	ReadStatus
	(
		pDestAddr := ADR(OUT_State),
		sIPAddr := ParamIpAddress,
		tTimeout := ParamTimeOut,
		nTcpPort := ParamTcpPort,
		nQuantity := 1,
		nMBAddr := 2,
		cbLength := SIZEOF(OUT_State),
		ClockRead := ClockRead AND MesDataExd.MesData.MesCP_Read,
		nUnitID := ParamUnitID
	);
	
	R_TrigState(CLK := OUT_State AND TpUpdate.Q);
	F_TrigState(CLK := OUT_State AND TpUpdate.Q);
	
	IF R_TrigState.Q THEN
		TimeStart := TIME();
	END_IF
	IF F_TrigState.Q  THEN
		TimeNotStart := TIME();
		OUT_WorkingHr := OUT_WorkingHr + (TimeNotStart-TimeStart);
	END_IF
END_IF
END_METHOD

METHOD M_Write : BOOL
VAR_INPUT
END_VAR
VAR
	WordToWrite		: WORD;
	AX_Addr			: ARRAY[1..3] OF UINT :=[1, 2, 3];
	
END_VAR

WordToWrite := REAL_TO_WORD(IN_SetptTemp*10.0);

Trig_CmdStart(CLK  := IN_CmdStart);
Trig_CmdStop(CLK  := IN_CmdStop);	
Trig_CmdReset(CLk := IN_CmdReset_L);

TP_MaintainStart(IN := Trig_CmdStart.Q OR Trig_CmdStop.Q OR Trig_CmdReset.Q, PT := ParamMaintainPulse);
R_TrigWriteCmd(CLK := TP_MaintainStart.Q);


IF Trig_CmdStart.Q THEN
	BlockToWrite := 1;
END_IF

IF Trig_CmdStop.Q THEN
	BlockToWrite := 0;
END_IF

IF Trig_CmdReset.Q THEN
	BlockToWrite := 2;
END_IF

WriteSetpt
(
	InputWord := (WordToWrite),
	sIPAddr := ParamIpAddress,
	tTimeout := ParamTimeOut,
	nTCPport := ParamTcpPort,
	nMBAddr := 0,
	cbLength := SIZEOF(WordToWrite),
	nQuantity := 1,
	nUnitID := ParamUnitID,
	WriteCmd := ClockWrite AND MesDataExd.Mesdata.MesCP_Write
);


WriteCmd
(
	bValue := TP_MaintainStart.Q,
	sIPAddr := ParamIpAddress,
	tTimeout := ParamTimeOut,
	nTCPport := ParamTcpPort,
	nMBAddr := BlockToWrite,
	nUnitID := ParamUnitID,
	WriteCmd := R_TrigWriteCmd.Q OR F_TrigWriteCmd.Q AND MesDataExd.Mesdata.MesCP_Write,
);
END_METHOD

END_FUNCTION_BLOCK

// ---- 01_Equipement_Library/HVAC/FB_HVAC_MADI.TcPOU
FUNCTION_BLOCK FB_HVAC_MADI EXTENDS FB_HVAC_Base
VAR_INPUT PERSISTENT
	ParamTempoComAlarm						: TIME 		:= T#10S ; 	(* (s) Config : Tempo to detect LOC Alarm	*)
	{attribute 'OPC.UA.DA' := '1'}                                  
	ParamIpAddress							: STRING;				(* IP Address                               *)
	{attribute 'OPC.UA.DA' := '1'}                                  
	ParamUnitID								: BYTE  	:= 1 ; 		(* Modbus Unit ID                           *)
	{attribute 'OPC.UA.DA' := '1'}                                 
	ParamTcpPort							: UINT 		:= 502;		(* Modbus TCP Port                          *)
	ParamPriority							: UINT;					(* Level of priority in the HVAC pool       *)
	
	ParamTimeOut							: TIME 		:= T#3S;	(* Modbus Timeout                           *)


	
END_VAR

VAR_INPUT	
	IN_SetptTemp				AT %Q*		: REAL:=22;
	IN_SetptHygro							: REAL;
	IN_CmdStart								: BOOL;
	IN_CmdStop								: BOOL;
	IN_CmdReset								: BOOL;

	IN_CmdReleaseStop_OPC					: BOOL ; // Manual Cmd. Non prioritaire sur le mode auto. 
	IN_CmdStop_OPC							: BOOL ; // Manual Cmd .Prioriatire sur le mode auto . Dévérouillage seulement sur ordre de start manual.  
	
	MesDataExd					AT %Q*: HVAC_MADI;	
END_VAR

VAR
	
	//M_ALARMMANAGEMENT VARIABLES 
		TON_ComAlarm				: TON ; 												// Tempo before detecting loss of communication. 
	

	
		
	//M_READ VARIABLES//
		WriteSetpt						: ARRAY[1..2] OF  FB_ModbusWriteSingleRegister;
		WriteCmd						: ARRAY[1..2] OF  FB_ModbusWriteSingleCoil;
		ReadStatus						: FB_ModbusReadCoils;
		ReadStatus2						: FB_ModbusReadCoils;		
		ReadInteger						: FB_ModbusRead ; 
		

		
		
		MesBlock1_Temp					: ARRAY[0..14] OF  WORD ; 
		MesBlockInput 					: ARRAY[1..8] OF WORD ; 

		MesModbusAlarmCode					: ARRAY[1..2] OF  UDINT ; 
		MesModbusReadAlarm				:  ARRAY[1..2] OF  BOOL ; 
		
		
		MesModbsWriteAlarm				: ARRAY[1..4] OF BOOL ; 
		
		BlockToWrite				AT %Q*	: BOOL;		
	
		RS_StartStop					: RS ; 
		RS_ForceStopOPC					: RS;
	
		

		R_TrigState						: R_TRIG;
		F_TrigState						: F_TRIG;
		TimeStart						: TIME;
		TimeNotStart					: TIME;
		
END_VAR
VAR_OUTPUT PERSISTENT
	          			
END_VAR

METHOD M_AlarmManagement : BOOL
VAR_INPUT
END_VAR

VAR
	FB_AlarmCodeManager			: FB_AlarmCodeManager ;
	CMWarning: BOOL;
	CMAlarm: BOOL;
	MesWarningCom: BOOL;
	WriteAlarm: BOOL;
END_VAR
		CMWarning 		:= MesModbusReadAlarm[1] OR MesModbusReadAlarm[2];
		CMAlarm			:= MesModbusReadAlarm[1] AND MesModbusReadAlarm[2];
		
		WriteAlarm		:= MesModbsWriteAlarm[1] OR MesModbsWriteAlarm[2] OR MesModbsWriteAlarm[3] OR MesModbsWriteAlarm[4] ;
		
	// Warning
	MesWarningCom 		:= CMWarning ; 											//
	//Alarm
	TON_ComAlarm(IN:= CMAlarm, PT:= ParamTempoComAlarm, Q=>MesDataExd.MesData.MesAlarmCom) ;	 	


	FB_AlarmCodeManager(
		bAlarm1			:= MesDataExd.MesAlarmsSynthesis, 	// HVAC Alarm Synthesis 
		bAlarm2			:= MesDataExd.MesData.MesAlarmCom,			// Communication Alarm #COM
		bAlarm3			:= WriteAlarm,					// Write Alarm 
		bAlarm4			:= FALSE,						//
		bAlarm5			:= False,                       //
		bAlarm6			:= False,                       //
		bAlarm7			:= False,                       //
		bAlarm8			:= False,                       //
		bAlarm9			:= FALSE,						//
		bAlarm10		:= False,                       //
		bAlarm11		:= False,                       //
		bAlarm12		:= False,                       //
		bAlarm13		:= False,                       //
		bAlarm14		:= FALSE,						//
		bAlarm15		:= False,                       //
		wAlarmCode		=>MesDataExd.MesData.MesAlarmCode);       
		                                                
                                                        
// WARNING CODE //
	FB_AlarmCodeManager
(
 		bAlarm1			:= MesWarningCom,						// Communication warning  #COM
		bAlarm2			:= False,                               //
		bAlarm3			:= False,                               //
		bAlarm4			:= False,                               //
		bAlarm5			:= False,                               //
		bAlarm6			:= False,                               //
		bAlarm7			:= False,                               //
		bAlarm8			:= False,                               //
		bAlarm9			:= False,                               //
		bAlarm10		:= False,                               //
		bAlarm11		:= False,                               //
		bAlarm12		:= FALSE,								//
		bAlarm13		:= False,                               //
		bAlarm14		:= False,                               //
		bAlarm15		:= False,                               //
		wAlarmCode		=>MesDataExd.MesData.MesWarningCode				
);   


// ALARM WORD EQUIPEMNT 
(*
	FB_AlarmCodeManager
(
		bAlarm0			:= ,// General alarm compressor 1                 
 		bAlarm1			:= ,// General alarm compressor 2                 							   
		bAlarm2			:= ,// Low pressure alarm compressor 1                                           
		bAlarm3			:= ,// Low pressure alarm compressor 2                                           
		bAlarm4			:= ,// Air flow alarm                                                            
		bAlarm5			:= ,// Fan thermal overload alarm                                                
		bAlarm6			:= ,// Heater 1 overload alarm                                                   
		bAlarm7			:= ,// Heater 2 overload alarm                                                   
		bAlarm8			:= ,// Fire / smoke alarm                                                        
		bAlarm9			:= ,// Dirty filter alarm                                                        
		bAlarm10		:= ,// High room temperature alarm                                               
		bAlarm11		:= ,// Low room temperature alarm                                                
		bAlarm12		:= ,// High ambient humidity alarm                								
		bAlarm13		:= ,// Low ambient humidity alarm                                                
		bAlarm14		:= ,// Operating hour threshold alarm,compressor 1                               
		bAlarm15		:= ,//Operating hour threshold alarm,compressor 2                              
		wAlarmCode		=> 				
);   

	FB_AlarmCodeManager
(
		bAlarm0			:= ,// Fan operating hour threshold alarm     
 		bAlarm1			:= ,// Room temperature probe broken alarm    						   
		bAlarm2			:= ,// Recovery temperature probe broken alarm                             
		bAlarm3			:= ,// Outside temperature probe broken alarm                              
		bAlarm4			:= ,// Outlet temperature probe broken                                     
		bAlarm5			:= ,// Ambient humidity probe broken                                       
		bAlarm6			:= ,// Pressure probe 1 broken alarm                                       
		bAlarm7			:= ,// Pressure probe2 broken alarm                                        
		bAlarm8			:= ,// Cond. 1 temperature probe broken                                    
		bAlarm9			:= ,// Cond. 2 temperature probe broken                                    
		bAlarm10		:= ,// High current alarm in the humidifier                                
		bAlarm11		:= ,// Humidifier no water alarm                                           
		bAlarm12		:= ,// Humidifier no current alarm            							
		bAlarm13		:= ,// Clock board broken alarm                                            
		bAlarm14		:= ,// High pressure alarm circuit 1                                       
		bAlarm15		:= ,//OHigh pressure alarm circuit 2                                     
		wAlarmCode		=> 				
);   

	FB_AlarmCodeManager
(
		bAlarm0			:= ,// Flood alarm                                
 		bAlarm1			:= ,// Auxiliary alarm                            					   
		bAlarm2			:= ,// Thermal overload and high pressure , comp 1                           
		bAlarm3			:= ,// Operating hour threshold alarm, humidifier                            
		bAlarm4			:= ,// Thermal overload and high pressure, comp 2                            
		bAlarm5			:= ,// Condenser fan 1 thermal overload                                      
		bAlarm6			:= ,// Condenser fan 1 thermal overload                                      
		bAlarm7			:= ,// Water flow alarm                                                      
		bAlarm8			:= ,// Driver 1 disconnected                                                 
		bAlarm9			:= ,// Driver 2 disconnected                                                 
		bAlarm10		:= ,// Cylinder maintenance mandatory                                        
		bAlarm11		:= ,// High conductivity alarm                                               
		bAlarm12		:= ,// Drain alarm humidifier                     						
		bAlarm13		:= ,// Full Cylinder alarm                                                   
		bAlarm14		:= ,// Foam in humidifier                                                    
		bAlarm15		:= ,// Cylinder exhausted                                                 
		wAlarmCode		=> 				
);   









*)
END_METHOD

METHOD M_CP : BOOL
VAR_INPUT
END_VAR


SUPER^.M_CP() ; 




Trig_Cmd_Read(CLK:=IN_CmdToggleRead);
Trig_Cmd_Write(CLK:=IN_CmdToggleWrite);
	
IF Trig_Cmd_Read.Q THEN
	IN_CmdToggleRead := FALSE;
	MesDataExd.MesData.MesCP_Read := NOT MesDataExd.MesData.MesCP_Read;
END_IF


IF Trig_Cmd_Write.Q THEN
	IN_CmdToggleWrite := FALSE;
	MesDataExd.MesData.MesCP_Write := NOT MesDataExd.MesData.MesCP_Write;
END_IF
END_METHOD

METHOD M_Evaluate : BOOL
VAR_INPUT
END_VAR
// Evaluate 
R_TrigState(CLK := MesDataExd.MesData.MesOn AND TpUpdate.Q);
F_TrigState(CLK := MesDataExd.MesData.MesOn AND TpUpdate.Q);

IF R_TrigState.Q THEN
	TimeStart := TIME();
END_IF
IF F_TrigState.Q  THEN
	TimeNotStart := TIME();
	WorkingHr := WorkingHr + (TimeNotStart-TimeStart);
	
END_IF

MesDataExd.MesData.MesWorkingHr := TIME_TO_REAL(WorkingHr) / 1000 ;
END_METHOD

METHOD M_Read : BOOL
VAR
		MW 					: FB_MergeWordsToDint; 
	MesAlarm1: WORD;
	MesAlarm3: WORD;
	MesAlarm2: WORD;
	MesData: INT;
END_VAR
//INITIALIZING MODBUS REQUESTS //
	ReadInteger(Reset:= CmdClearFault_G  ,sIPAddr:=ParamIpAddress, tTimeout:= ParamTimeout,nTcpPort:=502);

// CP-Read / Write 


IF MesDataExd.MesData.MesCP_Read  THEN	


	ReadInteger(
		nQuantity		:= 15, 
		nMBAddr			:= 1, 
		nUnitID			:= ParamUnitID,
		cbLength		:= SIZEOF(MesBlock1_Temp) , 
		pDestAddr		:= ADR(MesBlock1_Temp) ,
		ClockRead		:= MesDataExd.MesData.MesCP_Read AND ClockRead ,
		ModbusReadAlarm	=>	MesModbusReadAlarm[1] , 
		ErrorId			=> MesModbusAlarmCode[1]);	
		
				
	ReadStatus
	(
		pDestAddr := ADR(MesBlockInput),
		sIPAddr := ParamIpAddress,
		tTimeout := ParamTimeOut,
		nTcpPort := ParamTcpPort,
		nQuantity := 115,
		nMBAddr := 28,
		cbLength := SIZEOF(MesBlockInput),
		ClockRead := ClockRead and MesDataExd.MesData.MesCP_Read,
		nUnitID := ParamUnitID,
		Reset :=CmdClearFault_G  , 
		ModbusReadAlarm=>MesModbusReadAlarm[2] ,
		ErrorId =>MesModbusAlarmCode[2]
	);

	
	///
	MW(WORD_STRONG:= MesBlock1_Temp[ 0], 	SIGNED:=TRUE, FIX:=1 , SIZE:=1, VAR_OUT := MesDataExd.MesHygro_Amb);
	MW(WORD_STRONG:= MesBlock1_Temp[ 1], 	SIGNED:=TRUE, FIX:=1 , SIZE:=1, VAR_OUT := MesDataExd.MesPressure1);
	//MW(WORD_STRONG:= MesBlock1_Temp[ 2], 	SIGNED:=TRUE, FIX:=1 , SIZE:=1, VAR_OUT := MesDataExd.MesData.MesPressure2);
	MW(WORD_STRONG:= MesBlock1_Temp[ 3], 	SIGNED:=TRUE, FIX:=1 , SIZE:=1, VAR_OUT := MesDataExd.MesTemp_Room);
	MW(WORD_STRONG:= MesBlock1_Temp[ 4], 	SIGNED:=TRUE, FIX:=1 , SIZE:=1, VAR_OUT := MesDataExd.MesTemp_Outlet);
	MW(WORD_STRONG:= MesBlock1_Temp[ 5], 	SIGNED:=TRUE, FIX:=1 , SIZE:=1, VAR_OUT := MesDataExd.MesTemp_Outside);
	//MW(WORD_STRONG:= MesBlock1_Temp[ 6], 	SIGNED:=TRUE, FIX:=1 , SIZE:=1, VAR_OUT := MesDataExd.MesData.MesCondensing1);
	//MW(WORD_STRONG:= MesBlock1_Temp[ 7], 	SIGNED:=TRUE, FIX:=1 , SIZE:=1, VAR_OUT := MesDataExd.MesData.MesCondensing2);
	//MW(WORD_STRONG:= MesBlock1_Temp[ 8], 	SIGNED:=TRUE, FIX:=1 , SIZE:=1, VAR_OUT := MesDataExd.MesData.MesWaterRecov);
	MW(WORD_STRONG:= MesBlock1_Temp[ 9], 	SIGNED:=TRUE, FIX:=1 , SIZE:=1, VAR_OUT := MesDataExd.MesData.MesSetptTemp);
	MW(WORD_STRONG:= MesBlock1_Temp[ 10], 	SIGNED:=TRUE, FIX:=1 , SIZE:=1, VAR_OUT := MesDataExd.MesSetptTempmin);
	MW(WORD_STRONG:= MesBlock1_Temp[ 11], 	SIGNED:=TRUE, FIX:=1 , SIZE:=1, VAR_OUT := MesDataExd.MesSetptTempmax);
	MW(WORD_STRONG:= MesBlock1_Temp[ 12], 	SIGNED:=TRUE, FIX:=1 , SIZE:=1, VAR_OUT := MesDataExd.MesData.MesSetptHygro);
	MW(WORD_STRONG:= MesBlock1_Temp[ 13], 	SIGNED:=TRUE, FIX:=1 , SIZE:=1, VAR_OUT := MesDataExd.MesSetptHygromin);
	MW(WORD_STRONG:= MesBlock1_Temp[ 14], 	SIGNED:=TRUE, FIX:=1 , SIZE:=1, VAR_OUT := MesDataExd.MesSetptHygromax);
	
	
	MesDataExd.MesAlarm1 := MesBlockInput[1] ; 
	MesDataExd.MesAlarm2 := MesBlockInput[2] ; 
	MesDataExd.MesAlarm3 := MesBlockInput[3] ; 
	MesDataExd.MesAlarm3 := SHR(SHL(MesDataExd.MesAlarm3,8),8 ) ; 	// Keep only fist 8 bits . 
	MesDataExd.MesAlarm3.8 := MesBlockInput[7].0  ; 		// Driver 1 disconnected
	MesDataExd.MesAlarm3.9 := MesBlockInput[7].1  ; 		// Driver 2 disconnected
	MesDataExd.MesAlarm3.10 := MesBlockInput[7].2  ; 		// Cylinder maintenance mandatory
	MesDataExd.MesAlarm3.11 := MesBlockInput[7].4  ; 		// High conductivity alarm
	MesDataExd.MesAlarm3.12 := MesBlockInput[7].7  ; 		// Drain alarm humidifier
	MesDataExd.MesAlarm3.13 := MesBlockInput[7].8  ; 		// Full Cylinder alarm
	MesDataExd.MesAlarm3.14 := MesBlockInput[7].10  ; 		// Foam in humidifier
	MesDataExd.MesAlarm3.15 := MesBlockInput[7].11  ; 		//  Cylinder exhausted 
	
	MesDataExd.MesData.MesOn 	:=   MesBlockInput[7].15 ; 
	MesDataExd.MesCooling 		:=   MesBlockInput[8].0 ; 
	MesDataExd.MesHeating 		:=   MesBlockInput[8].1 ; 

END_IF

MesDataExd.MesAlarmsSynthesis := (MesDataExd.MesAlarm1 OR MesDataExd.MesAlarm2 OR MesDataExd.MesAlarm3) > 0 ;
END_METHOD

METHOD M_Write : BOOL
VAR_INPUT
END_VAR
VAR
	WordToWrite		: WORD;
	
	WordToWrite2: WORD;
	CHECK: BOOL;
	WriteCmd1: BOOL;

END_VAR
WordToWrite := REAL_TO_WORD(IN_SetptTemp*10);	// FIX 1 
WordToWrite2 := REAL_TO_WORD(IN_SetptHygro*10);	// FIX 1 


// Write Setpoint Temp
WriteSetpt[1]
(
	InputWord := (WordToWrite),
	sIPAddr := ParamIpAddress,
	tTimeout := ParamTimeOut,
	nTCPport := ParamTcpPort,
	nMBAddr := 10,
	cbLength := SIZEOF(WordToWrite),
	nQuantity := 1,
	nUnitID := ParamUnitID,
	WriteCmd := ClockWrite AND MesDataExd.Mesdata.MesCP_Write,
	ModbusWriteAlarm=> MesModbsWriteAlarm[1] 
);

// Write Setpoint Hygro 

WriteSetpt[2]
(
	InputWord := (WordToWrite2),
	sIPAddr := ParamIpAddress,
	tTimeout := ParamTimeOut,
	nTCPport := ParamTcpPort,
	nMBAddr := 13,
	cbLength := SIZEOF(WordToWrite2),
	nQuantity := 1,
	nUnitID := ParamUnitID,
	WriteCmd := ClockWrite AND MesDataExd.Mesdata.MesCP_Write,
	ModbusWriteAlarm=> MesModbsWriteAlarm[2] 
);

//RS_ForceStopOPC(SET:= IN_CmdStop_OPC  , RESET1:= IN_CmdReleaseStop_OPC ) ; 

RS_StartStop(SET:= IN_CmdStart , RESET1:= IN_CmdStop OR IN_CmdStop_OPC) ; //RS_ForceStopOPC.Q1 ) ; // Force stop if manual mode stop. 


// Start Stop 
// WRITE ON CHANGE //
	// Detect if another status is already forced . 
	CHECK := RS_StartStop.Q1 <>MesDataExd.MesData.MesOn ; 

	WriteCmd1 			:=(CHECK AND  ClockWrite) AND MesDataExd.Mesdata.MesCP_Write  ; 
BlockToWrite		:= RS_StartStop.Q1 ;

WriteCmd[1]
(
	bValue :=  RS_StartStop.Q1, //TP_MaintainStart.Q,
	sIPAddr := ParamIpAddress,
	tTimeout := ParamTimeOut,
	nTCPport := ParamTcpPort,
	nMBAddr := 112,
	nUnitID := ParamUnitID,
	WriteCmd := WriteCmd1,
	ModbusWriteAlarm=> MesModbsWriteAlarm[3] 
);



// Reset . One reset every day . After MainMVCB close

Trig_CmdReset(CLk := IN_CmdReset  );
FTrig_CmdReset(CLk := A1_SUBMV.A1_MainMVCB.MesDataExd.MesData.MesOpened );


WriteCmd[2]
(
	bValue := FTrig_CmdReset.Q OR IN_CmdReset OR (CalLocalTimeStruct.wHour = 6 AND CalLocalTimeStruct.wMinute = 0 AND (CalLocalTimeStruct.wSecond >= 0 AND CalLocalTimeStruct.wSecond <=  5)),
	sIPAddr := ParamIpAddress,
	tTimeout := ParamTimeOut,
	nTCPport := ParamTcpPort,
	nMBAddr := 123,
	nUnitID := ParamUnitID,
	WriteCmd :=  MesDataExd.Mesdata.MesCP_Write AND (NOT ClockWrite OR (Trig_CmdReset.Q ) OR FTrig_CmdReset.Q) ,
	ModbusWriteAlarm=> MesModbsWriteAlarm[4] 
);
END_METHOD

END_FUNCTION_BLOCK

// ---- 01_Equipement_Library/Inverter/FB_INV_ABB_PVS175TL.TcPOU
FUNCTION_BLOCK FB_INV_ABB_PVS175TL EXTENDS FB_INV_Base


VAR_INPUT PERSISTENT
	{attribute 'OPC.UA.DA' := '1'} 
	ParamTcpPort				: UINT	:= 502 ;		(* Modbus TCP port										*)	
	                                                	                                            			
	{attribute 'OPC.UA.DA' := '1'}                  	                                            			
	ParamIPAddress				: STRING; 				(* (NA)Config: IP Adress of PV INverter	    			*)
	{attribute 'OPC.UA.DA' := '1'}                  	                                            			
	ParamUnitID 				: BYTE; 				(* (NA)   SMA Modbus Unit ID.               			*)
	ParamNumInv					: BYTE;             	(* (NA) Inverter Index                           			*)
	ParamNumPTR					: UINT		:= 1;		(* (NA) number of the SPP								*)
	ParamTime_DeviationAlarm	: TIME 		:= T#1H;	(* (h) TIME where P is far FROM average before alarm 	*)
	ParamP_DeviationAlarm		: REAL		:= 0.8;		(* (%) deviation where P is considered far from average *)
	ParamPdcNom					: REAL;		(* (kW) DC nominal power *)
END_VAR

VAR_INPUT 
	// Parameters of the Object (instance specific) 
	AcknowledgeOrder			: BOOL ;			(* Acknowledge fault										*)
	ParamNbInv					: WORD ;			(* (NA) Nb of inverters per inverter                        *)
	                                               
	ParamOptionActivated		: WORD ;			(* (NA) Option available on the inverter                    *)
	                                             
	ParamPRamp					:  REAL:= 0 ;		(* (s) duration of the ramp from setpoint to setpoint       *)
	ParamQRamp					:  REAL:= 0 ;		(* (s) duration of the ramp from setpoint to setpoint       *)
	ParamPfRamp					:  REAL:= 0 ;		(* (s) duration of the ramp from setpoint to setpoint       *)
                                                                                                                
	IN_MesAcCbOpen_IO			:  BOOL ; 			(* Retour cablé Physique des contacteur AC des onduleurs	*)
	Cmd_SwitchOff				:  BOOL ;		    (* etat de DO cablé sur les onduleurs pour les eteindres    *)
	
	IN_SetptP					: REAL;
	IN_SetptQ					: REAL;
	IN_SetptCosPhi				: REAL;
	
	MesDataExd			AT %Q*	: INV_ABB_PVS;
END_VAR



VAR
	//M_Acknowledge
		
	// M_ALARMMNGMT VARIABLES //
	
		AX_TON_String				: ARRAY[1..12] OF TON;
		
	// M_READ VARIABLES//
		
		ModbusRead		   			: ARRAY[1..4] OF FB_ModbusRead ; 					// (NA) FB for Modbus Reading
		ModbusWrite	 	  			: ARRAY[1..2] OF FB_ModbusWrite ; 					// (NA) Functionnal Block for Writing Curtail limit through modbus	
		
		MesBlock_Temp 				: ARRAY[1..4] OF ARRAY[1..120]  OF WORD; 			// (NA) Temporary Block with multiple modbus reading (Caution : Double Word variables)
		MesModbusReadAlarm 		  	: ARRAY[1..4] OF BOOL ; 							// (NA) Modbus Read Alarm for all modbus frames		
		MesModbusAlarmCode			: ARRAY[1..4] OF UDINT;								// (NA) Modbus Read Alarm Code		
		MesModbusReadBusy			: ARRAY[1..4] OF BOOL;								// (NA) Modbus Read Busy  
		MesModbusReadCompleted		: ARRAY[1..4] OF BOOL;								// (NA) Modbus Read Completed
		

		MesModbusWriteAlarm		  	: ARRAY[1..2] OF BOOL ; 							// (NA) Modbus Read Alarm for all modbus frames		
		MesModbusWriteAlarmCode		: ARRAY[1..2] OF UDINT;								// (NA) Modbus Read Alarm Code		
		
		Trig_Midnight				: R_TRIG;
		Trig_Seconde				: R_TRIG;
		
	// M_CURTAIL VARIABLES //
	
		CmdPF_IO					: BOOL;
		CmdP_IO						: BOOL;
		CmdQ_IO						: BOOL;	
	
		LastCurtailMode				: BOOL:=TRUE ;				// Init at true, to force the first write on inverter
		MesCP_WriteCurtailMode		: BOOL ;
		CurtailModeValue_P			: DWORD ; 					// 1077 := WctlMan : Inverter set setpoint, 1079 := WCtlCom Inverter take the setpoint set by com (plc),303 := OFF
		CurtailModeValue_Q			: DWORD ;					// 303:=OFF,1075:= PFCtlCom,1074:= PFCtlMan,1072 VarCtlCom
		
		MesModbusWriteCode          : UDINT ; 					// (NA) Modbus Write Alarm Code 	
		MesModbusCurtailAlarm		: BOOL ;				   	// (NA) Modbus Write Curtail Alarm 
		
		InvQModeValue				: UINT ;					// Mode of Q power control : 1: Q mod, 2: PF mode, 3: Q(P)
		InvSetptQ					: REAL ;					// (kVAr) setpoint for the reactive power for each inverter
		
	
		InvSetptP					: REAL ;					// (kW) Setpoint for the active power for each inverter
		TEMP						: BOOL ;
		
		AX_CMD						: ARRAY[1..2] OF ARRAY[1..120] OF WORD;
		Trig_Reset					: R_TRIG;	
		
	// M_INIT //
		Code_Ctrl_Com 				: UINT := 1079 ;
		
		MesModbusCurtailInitAlarm 	: BOOL ;
		
	// M_STARTSTOP//
			                        	                            
		CmdStart					: BOOL;						// (NA) [P,H] External Start Command
		CmdStop 					: BOOL; 					// (NA) [P,H] External Stop Command. 
		TPStart						: TP ;						// (NA) TimeOut for start command
		TPStop						: TP ;						// (NA) TimeOut for stop command
		
		Trig_CmdP					: R_TRIG;
		Trig_CmdQ					: R_TRIG;
		Trig_CmdPF					: R_TRIG;

		TON_LowProd					: TON;
		
	// M_CP
		CalCP_Acknowledge			: BOOL ;
		//CalCP_CMD_SetPt				: BOOL; 	  // Write command start;
		CalCP_CMD_StartStop			: BOOL ; 		  // Write command start;
		CalCP_CMD_StartStopIO		: BOOL ; 		  // Write command start;
	// M_STATEMANAGER//
	
	//M_EXECUTE VARIABLES //
		TP_READ						: LTP ;			  //Tempo de cadencement FB Modbus
		RTrig						: R_Trig ; 		  //Front montant sur TP_READ.Q
		ReadBusy					: BOOL ;		 //FB Modbus en busy
		
	//EMULATOR VARIABLES //
		
END_VAR

METHOD M_AlarmManagement
//////////////////
// Manages IntelliGen Alarms
/////////////////

VAR 
	// Method local variables (reinitialized at each cycle) 
	FB_AlarmCodeManager : FB_AlarmCodeManager ; 

	KK					: BYTE;		// For Loop 
	
	ComWarning			: BOOL;		// Aggregated Wcommunication warning
	ComAlarm			: BOOL;		// Aggregated communication Alarm
	AX_Alarms			: ARRAY[1..4] of BOOL;
	LL: INT;
END_VAR
FOR KK := 1 TO 4 DO
	ComAlarm := ComAlarm AND ModbusRead[KK].ModbusReadAlarm;
	ComWarning := ComWarning OR ModbusRead[KK].ModbusReadAlarm;
END_FOR
ComAlarm := ComAlarm AND ModbusWrite[1].ModbusWriteAlarm AND ModbusWrite[2].ModbusWriteAlarm;
ComWarning := ComWarning OR ModbusWrite[1].ModbusWriteAlarm OR ModbusWrite[2].ModbusWriteAlarm ;

TON_ComAlarm	(IN := ComAlarm, PT := T#30S , Q=> MesDataExd.Mesdata.MesAlarmCom);
TON_ComWarning	(IN := ComWarning, PT := T#30S);

FOR KK := 1 TO 12 DO
	AX_TON_String[KK](in := MesDataExd.AX_STR[KK].MesIdc < 0.1, PT := T#24H);
END_FOR
FOR KK := 1 TO 4 DO
	FOR LL := 1 TO 3 DO
		AX_Alarms[KK] := AX_ALarms[KK] OR AX_TON_String[(KK-1)*3+LL].Q ;
	END_FOR
END_FOR

TON_LowProd(in := GVL_CFG.AX_PTR[ParamNumPTR].MesDataExd.MesP_Avg > MesDataExd.MesData.MesP / ParamP_DeviationAlarm AND GVL_CFG.AX_PTR[ParamNumPTR].MesDataExd.MesP_Avg > 10, pt := ParamTime_DeviationAlarm);

// ALARM CODE //
	FB_AlarmCodeManager(
		bAlarm1			:= MesDataExd.Mesdata.MesAlarmCom,  		// Communication Alarm                                   
		bAlarm2			:= NOT MesDataExd.CmdStart_Ack , 			// Stop order to Inv                                     
		bAlarm3			:= FALSE, //MesDataExd.MesData.MesStatus.7,			// Inverter is in Fault                                 
		bAlarm4			:= FALSE, //MesDataExd.MesEvent1>0, 					// Event1 alarm, check MesEvent1 word                        
		bAlarm5			:= FALSE, //MesDataExd.MesVndEventBitFld1> 1, 		// Inverter is derating : check Vendor event Bitfield1
		bAlarm6			:= FALSE, //MesDataExd.MesVndEventBitFld2>0, 		// Inverter is derating : check Vendor event Bitfield2 
		bAlarm7			:= FALSE, //MesDataExd.MesVndEventBitFld3>0,			// Alarm on Auxiliary devices                          
		bAlarm8			:= NOT MesdataExd.MesData.MesCP_Read, 		// Inverter data reading disabled                                  
		bAlarm9			:= NOT MesdataExd.MesData.MesCP_Write,		// Inverter data writing disabled                                  
		bAlarm10		:= AX_Alarms[1], 							// String 1 to 3 has not produced for 24h                             
		bAlarm11		:= AX_Alarms[2], 							// String 4 to 6 has not produced for 24h                             
		bAlarm12		:= AX_Alarms[3], 							// String 7 to 9 has not produced for 24h                             
		bAlarm13		:= AX_Alarms[4], 							// String 10 to 12 has not produced for 24h                           
		bAlarm14		:= TON_LowProd.Q, 							// Power is lower than average                           
		bAlarm15		:= FALSE, 									//                                                                        
		wAlarmCode		=>MesDataExd.MesData.MesAlarmCode);         

// ALARM CODE //
	FB_AlarmCodeManager(
		bAlarm1			:= AX_TON_String[1].Q, 						//	String 1 has not produced for 24h                   
		bAlarm2			:= AX_TON_String[2].Q,                      //	String 2 has not produced for 24h  
		bAlarm3			:= AX_TON_String[3].Q,                      //	String 3 has not produced for 24h 
		bAlarm4			:= AX_TON_String[4].Q,                      //	String 4 has not produced for 24h	     
		bAlarm5			:= AX_TON_String[5].Q,	                   	//	String 5 has not produced for 24h    
		bAlarm6			:= AX_TON_String[6].Q,                      //	String 6 has not produced for 24h 
		bAlarm7			:= AX_TON_String[7].Q,                      //	String 7 has not produced for 24h 
		bAlarm8			:= AX_TON_String[8].Q,                      //	String 8 has not produced for 24h            
		bAlarm9			:= AX_TON_String[9].Q,                      //	String 9 has not produced for 24h            
		bAlarm10		:= AX_TON_String[10].Q,                     //	String 10 has not produced for 24h             
		bAlarm11		:= AX_TON_String[11].Q,                     //	String 11 has not produced for 24h             
		bAlarm12		:= AX_TON_String[12].Q,                     //	String 12 has not produced for 24h             
		bAlarm13		:= FALSE,              
		bAlarm14		:= FALSE,
		bAlarm15		:= FALSE,                   
		wAlarmCode		=>MesDataExd.MesData.MesAlarmCode2);                                                    

// WARNING CODE //
	FB_AlarmCodeManager(
 		bAlarm1			:= FALSE,									//
		bAlarm2			:= FALSE,									//
		bAlarm3			:= FALSE,									//
		bAlarm4			:= FALSE,									//
		bAlarm5			:= FALSE,									//
		bAlarm6			:= FALSE,									//
		bAlarm7			:= FALSE,									//
		bAlarm8			:= FALSE,									//
		bAlarm9			:= FALSE,									//
		bAlarm10		:= FALSE,									//
		bAlarm11		:= FALSE,									//
		bAlarm12		:= FALSE,									//
		bAlarm13		:= FALSE,                                   //
		bAlarm14		:= FALSE,                                   //
		bAlarm15		:= TON_ComWarning.Q, 						// One or more error, communication frames for the past 30 seconds #COM
		wAlarmCode		=>MesDataExd.MesData.MesWarningCode);	
		
(*

	FB_AlarmCodeManager(
 		bAlarm1			:= FALSE,	//Off (OFF)
		bAlarm2			:= FALSE,	//Sleeping (SLEEPING)
		bAlarm3			:= FALSE,	//Starting (STARTING)
		bAlarm4			:= FALSE,	//MPPT
		bAlarm5			:= FALSE,	//Throttled (THROTTLED)
		bAlarm6			:= FALSE,	//Shutting down (SHUTTING_DOWN)
		bAlarm7			:= FALSE,	//Fault (FAULT)
		bAlarm8			:= FALSE,	//Standby (STANDBY)
		bAlarm9			:= FALSE,	//
		bAlarm10		:= FALSE,	//
		bAlarm11		:= FALSE,	//
		bAlarm12		:= FALSE,	//
		bAlarm13		:= FALSE,   //
		bAlarm14		:= FALSE,   //
		bAlarm15		:= FALSE, 	//
		wAlarmCode		=>MesDataExd.MesData.MesIDState);	
		

	FB_AlarmCodeManager(
  		bAlarm0			:= FALSE,	//Ground fault (GROUND_FAULT)
		bAlarm1			:= FALSE,	//DC over voltage (DC_OVER_VOLT)
		bAlarm2			:= FALSE,	//
		bAlarm3			:= FALSE,	//
		bAlarm4			:= FALSE,	//Grid shutdown (GRID_DISCONNECT)
		bAlarm5			:= FALSE,	//
		bAlarm6			:= FALSE,	//Manual shutdown (MANUAL_SHUTDOWN)
		bAlarm7			:= FALSE,	//Over temperature (OVER_TEMP)
		bAlarm8			:= FALSE,	//Frequency above limit (OVER_FREQUENCY)
		bAlarm9			:= FALSE,	//Frequency under limit (UNDER_FREQUENCY)
		bAlarm10		:= FALSE,	//AC Voltage above limit (AC_OVER_VOLT)
		bAlarm11		:= FALSE,	//AC Voltage under limit (AC_UNDER_VOLT)
		bAlarm12		:= FALSE,	//Under temperature (UNDER_TEMP)
		bAlarm13		:= FALSE,   //
		bAlarm14		:= FALSE,   //Generic Memory or Communication error (internal) (MEMORY_LOSS)
		bAlarm15		:= FALSE, 	//Hardware test failure (HW_TEST_FAILURE)
		wAlarmCode		=>MesDataExd.MesData.MesEvent1);		
		

	FB_AlarmCodeManager(
  		bAlarm0			:= FALSE,	//Power curtailment from external command (NOTE: Asserted also for limitation from capability together with bit 12).
		bAlarm1			:= FALSE,	//Power limitation from Frequency-Watt
		bAlarm2			:= FALSE,	//Power limitation from high average grid voltage
		bAlarm3			:= FALSE,	//Power limitation from anti-islanding protection
		bAlarm4			:= FALSE,	//Power limitation from grid current rating limitation
		bAlarm5			:= FALSE,	//Power limitation for high temperature
		bAlarm6			:= FALSE,	//Power limitation for high DC voltage
		bAlarm7			:= FALSE,	//Reserved
		bAlarm8			:= FALSE,	//Power limitation from ramp-rate (connection ramp)
		bAlarm9			:= FALSE,	//Power limitation from momentary cessation
		bAlarm10		:= FALSE,	//Power limitation from ramp-rate (normal ramp-up)
		bAlarm11		:= FALSE,	//Power limitation from Volt-Watt
		bAlarm12		:= FALSE,	//Power limitation from capability (rating)
		bAlarm13		:= FALSE,   //
		bAlarm14		:= FALSE,   //
		bAlarm15		:= FALSE, 	//
		wAlarmCode		=>MesDataExd.MesData.MesVndEventBitFld1);		
		

	FB_AlarmCodeManager(
  		bAlarm0			:= FALSE,	//Power limitation for high temperature    
		bAlarm1			:= FALSE,	//Power limitation for high DC voltage     
		bAlarm2			:= FALSE,	//Power limitation from capability (rating)
		bAlarm3			:= FALSE,	//
		bAlarm4			:= FALSE,	//
		bAlarm5			:= FALSE,	//
		bAlarm6			:= FALSE,	//
		bAlarm7			:= FALSE,	//
		bAlarm8			:= FALSE,	//
		bAlarm9			:= FALSE,	//
		bAlarm10		:= FALSE,	//
		bAlarm11		:= FALSE,	//
		bAlarm12		:= FALSE,	//
		bAlarm13		:= FALSE,   //
		bAlarm14		:= FALSE,   //
		bAlarm15		:= FALSE, 	//
		wAlarmCode		=>MesDataExd.MesData.MesVndEventBitFld2);	
		

	FB_AlarmCodeManager(
  		bAlarm0			:= FALSE,	//Fan fault
		bAlarm1			:= FALSE,	//Statistics memory fault
		bAlarm2			:= FALSE,	//RTC clock not set
		bAlarm3			:= FALSE,	//Reserved
		bAlarm4			:= FALSE,	//RTC low battery fault
		bAlarm5			:= FALSE,	//RTC quartz fault
		bAlarm6			:= FALSE,	//
		bAlarm7			:= FALSE,	//
		bAlarm8			:= FALSE,	//
		bAlarm9			:= FALSE,	//
		bAlarm10		:= FALSE,	//
		bAlarm11		:= FALSE,	//
		bAlarm12		:= FALSE,	//
		bAlarm13		:= FALSE,   //
		bAlarm14		:= FALSE,   //
		bAlarm15		:= FALSE, 	//
		wAlarmCode		=>MesDataExd.MesData.MesVndEventBitFld3);

		*)
END_METHOD

METHOD M_CP
//////////////////
//  Emulator
/////////////////

VAR 
	// Method local variables (reinitialized at each cycle) 
	MesOpState : BOOL;
END_VAR


SUPER^.M_CP() ; 




Trig_Cmd_Read(CLK:=IN_CmdToggleRead);
Trig_Cmd_Write(CLK:=IN_CmdToggleWrite);
	
IF Trig_Cmd_Read.Q THEN
	IN_CmdToggleRead := FALSE;
	MesDataExd.MesData.MesCP_Read := NOT MesDataExd.MesData.MesCP_Read;
END_IF


IF Trig_Cmd_Write.Q THEN
	IN_CmdToggleWrite := FALSE;
	MesDataExd.MesData.MesCP_Write := NOT MesDataExd.MesData.MesCP_Write;
END_IF
END_METHOD

{attribute 'object_name' := 'M_Curtail'}
METHOD M_Curtail
//////////////////
// Write Curtail Command through modbus to PV inverters.  
//////////////////
VAR 

	AX_ADDR 	: ARRAY[1..2] OF UINT := [40230 , 41356 ];
	AX_QTY 		: ARRAY[1..2] OF BYTE := [21	, 1];
	AX_UnitID 	: ARRAY[1..2] OF BYTE := [1 	, 1];

END_VAR
IF MesDataExd.MesData.MesCP_Write THEN

	AX_CMD[1][1] := 0;														// Time Window for connect/disconnect
	AX_CMD[1][2] := 600;													// Timeout period for connect/disconnect.
	AX_CMD[1][3] := BOOL_TO_WORD(MesDataExd.CmdStart_Ack);					// Start Cmd
	AX_CMD[1][4] := REAL_TO_WORD(MesDataExd.MesData.OUT_SetptPLimit*1000/ParamPn);	// SetptP
	AX_CMD[1][5] := 0;														// Time Window for SetptP
	AX_CMD[1][6] := 600;													// Timeout for SetptP
	AX_CMD[1][7] := 0;														// Ramp time for SetptP
	AX_CMD[1][8] := BOOL_TO_WORD(MesDataExd.CmdP_Ack);						// Enable / disable SetptP
	AX_Cmd[1][9] := REAL_TO_WORD(MesDataExd.OUT_SetptCosPhi*10000);			// Power factor setpoint
	AX_Cmd[1][10] := 0;														// Time Window for PF
	AX_CMD[1][11] := 600;													// Timeout for PF
	AX_CMD[1][12] := 0;														// Ramp time for PF
	AX_Cmd[1][13] := BOOL_TO_WORD(MesDataExd.CmdPF_Ack);					// PF Setpoint Enabled
	AX_Cmd[1][14] := REAL_TO_WORD(MesDataExd.MesData.OUT_SetptQ*1000/ParamPn);	// SetptQ
	AX_Cmd[1][17] := 0;														// Time Window for Q
	AX_CMD[1][18] := 600;													// Timeout for Q
	AX_CMD[1][19] := 0;														// Ramp time for Q
	AX_CMD[1][20] := BOOL_TO_WORD(MesDataExd.CmdQ_Ack);						// Q Setpoint Enabled
	AX_CMD[1][21] := 1;													// 
	
	
	AX_Cmd[2][1] := BOOL_TO_WORD(Trig_Reset.Q);							// Cmd Reset
	
	ModbusWrite[1]
	(
		pSrcAddr := ADR(AX_CMD[1]),
		sIPAddr := ParamIPAddress,
		tTimeout := ParamTimeout,
		nTCPport := ParamTCPPort,
		nMBAddr := AX_ADDR[1],
		cbLength := SIZEOF(AX_CMD[1]),
		nQuantity := AX_QTY[1],
		nUnitID := AX_UnitId[1],
		WriteCmd := ClockWrite,
		ModbusWriteAlarm => MesModbusWriteAlarm[1]
	);

END_IF
END_METHOD

METHOD M_Evaluate
VAR_INPUT
END_VAR
MesDataExd.MesData.ParamPn := ParamPn;

MesDataExd.MesData.MesCurtl := MesDataExd.MesData.MesState_Inv.5;

MesDataExd.MesData.OUT_SetptP := MIN(IN_SetptP, ParamPn);
MesDataExd.MesData.OUT_SetptQ := MIN(ParamPn, MAX(-ParamPn, IN_SetptQ));
MesDataExd.OUT_SetptCosPhi := IN_SetptCosPhi;

Trig_Midnight(clk := CalLocalTimeStruct.wHour=0);
Trig_Seconde(clk := CalLocalTimeStruct.wMilliseconds<500);

IF Trig_Midnight.Q THEN
	MesDataExd.MesEacDay := 0;
END_IF
IF Trig_Seconde.Q THEN
	MesDataExd.MesEacDay := MesDataExd.MesEacDay + MesDataExd.MesData.MesP/3600;
END_IF
END_METHOD

METHOD M_Execute
//////////////////
//  Method Calls 
/////////////////

VAR 
	// Method local variables (reinitialized at each cycle) 

END_VAR
IF  bInit THEN
	M_Init();
END_IF


SUPER^.M_Execute() ;
END_METHOD

{attribute 'object_name' := 'M_Read'}
METHOD M_Read
//////////
// Read Method for SMA : Modbus reading
//////////
VAR
	// Method local variables (reinitialized at each cycle) 
	MW 					: FB_MergeWordsToDint; 
	

	KK					: BYTE;						 // Index to loop over modbus blocks. 	
	JJ					: BYTE;						// Index loop over Number of SB
	
	
	AX_ADDR				: ARRAY[1..4] OF UINT := [40072,	40184, 	41110, 	41231];
	AX_QTY				: ARRAY[1..4] OF UINT := [47, 		43,		120,	120];
	AX_UnitId			: ARRAY[1..4] OF BYTE := [1, 		1, 		1, 		1];
	
	MesStatus: UINT;

END_VAR
IF MesDataExd.MesData.MesCP_Read THEN

	//INITIALIZING MODBUS REQUESTS //
	FOR KK := 1 TO 4 DO
		ModbusRead[KK] 
		(
			pDestAddr := ADR(MesBlock_Temp[KK]),
			sIPAddr := ParamIPAddress,
			tTimeout := ParamTimeout,
			nQuantity := AX_QTY[KK],
			ntcpport := ParamTCPPort,
			nMBAddr := AX_ADDR[KK],
			nUnitID := AX_UnitId[KK],
			cbLength := SIZEOF(MesBlock_Temp[KK]),
			ClockRead := ClockRead AND MesdataExd.MesData.MesCP_Read,
			Reset := CmdClearFault_G OR IN_CmdReset_L,
			ErrorId => MesModbusAlarmCode[KK],
			ModbusReadAlarm => MesModbusReadAlarm[KK],
			Busy => MesModbusReadBusy[KK]	
		);
	END_FOR
	
	
	MW( WORD_STRONG:= MesBlock_Temp[1][ 1], SIZE := 1, FIX := 1, SIGNED := FALSE,	VAR_OUT:=MesDataExd.MesData.MesI);
	MW( WORD_STRONG:= MesBlock_Temp[1][ 2], SIZE := 1, FIX := 1, SIGNED := FALSE,	VAR_OUT:=MesDataExd.MesI1);
	MW( WORD_STRONG:= MesBlock_Temp[1][ 3], SIZE := 1, FIX := 1, SIGNED := FALSE,	VAR_OUT:=MesDataExd.MesI2);
	MW( WORD_STRONG:= MesBlock_Temp[1][ 4], SIZE := 1, FIX := 1, SIGNED := FALSE,	VAR_OUT:=MesDataExd.MesI3);
	MW( WORD_STRONG:= MesBlock_Temp[1][ 6], SIZE := 1, FIX := 1, SIGNED := FALSE,	VAR_OUT:=MesDataExd.MesU12);
	MW( WORD_STRONG:= MesBlock_Temp[1][ 7], SIZE := 1, FIX := 1, SIGNED := FALSE,	VAR_OUT:=MesDataExd.MesU23);
	MW( WORD_STRONG:= MesBlock_Temp[1][ 8], SIZE := 1, FIX := 1, SIGNED := FALSE,	VAR_OUT:=MesDataExd.MesU31);;
	MW( WORD_STRONG:= MesBlock_Temp[1][ 9], SIZE := 1, FIX := 1, SIGNED := FALSE,	VAR_OUT:=MesDataExd.MesV1);
	MW( WORD_STRONG:= MesBlock_Temp[1][10], SIZE := 1, FIX := 1, SIGNED := FALSE,	VAR_OUT:=MesDataExd.MesV2);
	MW( WORD_STRONG:= MesBlock_Temp[1][11], SIZE := 1, FIX := 1, SIGNED := FALSE,	VAR_OUT:=MesDataExd.MesV3);
	MW( WORD_STRONG:= MesBlock_Temp[1][13], SIZE := 1, FIX := 2, SIGNED := TRUE,	VAR_OUT:=MesDataExd.MesData.MesP);
	MW( WORD_STRONG:= MesBlock_Temp[1][15], SIZE := 1, FIX := 2, SIGNED := FALSE,	VAR_OUT:=MesDataExd.MesData.MesFreq);
	MW( WORD_STRONG:= MesBlock_Temp[1][19], SIZE := 1, FIX := 2, SIGNED := TRUE,	VAR_OUT:=MesDataExd.MesData.MesQ);
	MW( WORD_STRONG:= MesBlock_Temp[1][21], SIZE := 1, FIX := 4, SIGNED := FALSE,	VAR_OUT:=MesDataExd.MesPF);
	MW( WORD_STRONG:= MesBlock_Temp[1][26], SIZE := 1, FIX := 1, SIGNED := FALSE,	VAR_OUT:=MesDataExd.MesData.MesIdc);
	MW( WORD_STRONG:= MesBlock_Temp[1][30], SIZE := 1, FIX := 2, SIGNED := TRUE,	VAR_OUT:=MesDataExd.MesData.MesPdc);
	MW( WORD_STRONG:= MesBlock_Temp[1][32], SIZE := 1, FIX := 1, SIGNED := FALSE,	VAR_OUT:=MesDataExd.MesTemp_AC_cab);
	MW( WORD_STRONG:= MesBlock_Temp[1][33], SIZE := 1, FIX := 1, SIGNED := FALSE,	VAR_OUT:=MesDataExd.MesTemp_HeatSink);
	
	MesDataExd.MesData.MesState_Inv						:= WORD_TO_UINT(MesBlock_Temp[1][37]);
	MesDataExd.MesState_InvWord.1 := MesBlock_Temp[1][37] = 1;
	MesDataExd.MesState_InvWord.2 := MesBlock_Temp[1][37] = 2;
	MesDataExd.MesState_InvWord.3 := MesBlock_Temp[1][37] = 3;
	MesDataExd.MesState_InvWord.4 := MesBlock_Temp[1][37] = 4;
	MesDataExd.MesState_InvWord.5 := MesBlock_Temp[1][37] = 5;
	MesDataExd.MesState_InvWord.6 := MesBlock_Temp[1][37] = 6;
	MesDataExd.MesState_InvWord.7 := MesBlock_Temp[1][37] = 7;
	MesDataExd.MesState_InvWord.8 := MesBlock_Temp[1][37] = 8;
	
	MesDataExd.MesVndOpeState 			:= WORD_TO_UINT(MesBlock_Temp[1][38]);
	MesDataExd.MesEvent1 				:= DWORD_TO_WORD(SHL(WORD_TO_DWORD(MesBlock_Temp[1][39]), 16) OR  MesBlock_Temp[1][40]);
	MesDataExd.MesEventBitFld2 			:= DWORD_TO_WORD(SHL(WORD_TO_DWORD(MesBlock_Temp[1][41]), 16) OR  MesBlock_Temp[1][42]);
	MesDataExd.MesVndEventBitFld1 		:= DWORD_TO_WORD(SHL(WORD_TO_DWORD(MesBlock_Temp[1][43]), 16) OR  MesBlock_Temp[1][44]);
	MesDataExd.MesVndEventBitFld2 		:= DWORD_TO_WORD(SHL(WORD_TO_DWORD(MesBlock_Temp[1][45]), 16) OR  MesBlock_Temp[1][46]);
	MesDataExd.MesVndEventBitFld3 		:= DWORD_TO_WORD(SHL(WORD_TO_DWORD(MesBlock_Temp[1][47]), 16) OR  MesBlock_Temp[1][48]);
	
	
	MEMCPY(destAddr := ADR(MesDataExd.MesEacTot), srcAddr := ADR(MesBlock_Temp[2][7]), n := 2);
	MEMCPY(destAddr := ADR(MesDataExd.MesEacTot)+SIZEOF(MesBlock_Temp[2][1]), srcAddr := ADR(MesBlock_Temp[2][6]), n := 2);
	MEMCPY(destAddr := ADR(MesDataExd.MesEacTot)+2*SIZEOF(MesBlock_Temp[2][1]), srcAddr := ADR(MesBlock_Temp[2][5]), n := 2);
	MEMCPY(destAddr := ADR(MesDataExd.MesEacTot)+3*SIZEOF(MesBlock_Temp[2][1]), srcAddr := ADR(MesBlock_Temp[2][4]), n := 2);
	
	
	
	MW( WORD_STRONG:= MesBlock_Temp[2][43], SIZE := 1, FIX := 0, SIGNED := FALSE,	VAR_OUT:=MesDataExd.MesData.MesInsuResistor);// kohms
	
	memcpy(destAddr := ADR(MesDataExd.MesGlobalEvt), srcAddr := ADR(MesBlock_Temp[3][1]), n := SIZEOF(MesBlock_Temp[3][1]));
	memcpy(destAddr := ADR(MesDataExd.MesGlobalEvt)+ SIZEOF(MesBlock_Temp[3][1]), srcAddr := ADR(MesBlock_Temp[3][2]), n := SIZEOF(MesBlock_Temp[3][2]));
	
	MW( WORD_STRONG:= MesBlock_Temp[3][ 14], SIZE := 1, FIX := 1, SIGNED := FALSE,	VAR_OUT:= MesDataExd.AX_STR[ 1].MesIdc);
	MW( WORD_STRONG:= MesBlock_Temp[3][ 15], SIZE := 1, FIX := 1, SIGNED := FALSE,	VAR_OUT:= MesDataExd.AX_STR[ 1].MesUdc);
	MW( WORD_STRONG:= MesBlock_Temp[3][ 16], SIZE := 1, FIX := 2, SIGNED := FALSE,	VAR_OUT:= MesDataExd.AX_STR[ 1].MesPdc);
	MW( WORD_STRONG:= MesBlock_Temp[3][ 34], SIZE := 1, FIX := 1, SIGNED := FALSE,	VAR_OUT:= MesDataExd.AX_STR[ 2].MesIdc);
	MW( WORD_STRONG:= MesBlock_Temp[3][ 35], SIZE := 1, FIX := 1, SIGNED := FALSE,	VAR_OUT:= MesDataExd.AX_STR[ 2].MesUdc);
	MW( WORD_STRONG:= MesBlock_Temp[3][ 36], SIZE := 1, FIX := 2, SIGNED := FALSE,	VAR_OUT:= MesDataExd.AX_STR[ 2].MesPdc);
	MW( WORD_STRONG:= MesBlock_Temp[3][ 54], SIZE := 1, FIX := 1, SIGNED := FALSE,	VAR_OUT:= MesDataExd.AX_STR[ 3].MesIdc);
	MW( WORD_STRONG:= MesBlock_Temp[3][ 55], SIZE := 1, FIX := 1, SIGNED := FALSE,	VAR_OUT:= MesDataExd.AX_STR[ 3].MesUdc);
	MW( WORD_STRONG:= MesBlock_Temp[3][ 56], SIZE := 1, FIX := 2, SIGNED := FALSE,	VAR_OUT:= MesDataExd.AX_STR[ 3].MesPdc);
	MW( WORD_STRONG:= MesBlock_Temp[3][ 74], SIZE := 1, FIX := 1, SIGNED := FALSE,	VAR_OUT:= MesDataExd.AX_STR[ 4].MesIdc);
	MW( WORD_STRONG:= MesBlock_Temp[3][ 75], SIZE := 1, FIX := 1, SIGNED := FALSE,	VAR_OUT:= MesDataExd.AX_STR[ 4].MesUdc);
	MW( WORD_STRONG:= MesBlock_Temp[3][ 76], SIZE := 1, FIX := 2, SIGNED := FALSE,	VAR_OUT:= MesDataExd.AX_STR[ 4].MesPdc);
	MW( WORD_STRONG:= MesBlock_Temp[3][ 94], SIZE := 1, FIX := 1, SIGNED := FALSE,	VAR_OUT:= MesDataExd.AX_STR[ 5].MesIdc);
	MW( WORD_STRONG:= MesBlock_Temp[3][ 95], SIZE := 1, FIX := 1, SIGNED := FALSE,	VAR_OUT:= MesDataExd.AX_STR[ 5].MesUdc);
	MW( WORD_STRONG:= MesBlock_Temp[3][ 96], SIZE := 1, FIX := 2, SIGNED := FALSE,	VAR_OUT:= MesDataExd.AX_STR[ 5].MesPdc);
	MW( WORD_STRONG:= MesBlock_Temp[3][114], SIZE := 1, FIX := 1, SIGNED := FALSE,	VAR_OUT:= MesDataExd.AX_STR[ 6].MesIdc);
	MW( WORD_STRONG:= MesBlock_Temp[3][115], SIZE := 1, FIX := 1, SIGNED := FALSE,	VAR_OUT:= MesDataExd.AX_STR[ 6].MesUdc);
	MW( WORD_STRONG:= MesBlock_Temp[3][116], SIZE := 1, FIX := 2, SIGNED := FALSE,	VAR_OUT:= MesDataExd.AX_STR[ 6].MesPdc);
	
	MW( WORD_STRONG:= MesBlock_Temp[4][ 13], SIZE := 1, FIX := 1, SIGNED := FALSE,	VAR_OUT:= MesDataExd.AX_STR[ 7].MesIdc);
	MW( WORD_STRONG:= MesBlock_Temp[4][ 14], SIZE := 1, FIX := 1, SIGNED := FALSE,	VAR_OUT:= MesDataExd.AX_STR[ 7].MesUdc);
	MW( WORD_STRONG:= MesBlock_Temp[4][ 15], SIZE := 1, FIX := 2, SIGNED := FALSE,	VAR_OUT:= MesDataExd.AX_STR[ 7].MesPdc);
	MW( WORD_STRONG:= MesBlock_Temp[4][ 33], SIZE := 1, FIX := 1, SIGNED := FALSE,	VAR_OUT:= MesDataExd.AX_STR[ 8].MesIdc);
	MW( WORD_STRONG:= MesBlock_Temp[4][ 34], SIZE := 1, FIX := 1, SIGNED := FALSE,	VAR_OUT:= MesDataExd.AX_STR[ 8].MesUdc);
	MW( WORD_STRONG:= MesBlock_Temp[4][ 35], SIZE := 1, FIX := 2, SIGNED := FALSE,	VAR_OUT:= MesDataExd.AX_STR[ 8].MesPdc);
	MW( WORD_STRONG:= MesBlock_Temp[4][ 53], SIZE := 1, FIX := 1, SIGNED := FALSE,	VAR_OUT:= MesDataExd.AX_STR[ 9].MesIdc);
	MW( WORD_STRONG:= MesBlock_Temp[4][ 54], SIZE := 1, FIX := 1, SIGNED := FALSE,	VAR_OUT:= MesDataExd.AX_STR[ 9].MesUdc);
	MW( WORD_STRONG:= MesBlock_Temp[4][ 55], SIZE := 1, FIX := 2, SIGNED := FALSE,	VAR_OUT:= MesDataExd.AX_STR[ 9].MesPdc);
	MW( WORD_STRONG:= MesBlock_Temp[4][ 73], SIZE := 1, FIX := 1, SIGNED := FALSE,	VAR_OUT:= MesDataExd.AX_STR[10].MesIdc);
	MW( WORD_STRONG:= MesBlock_Temp[4][ 74], SIZE := 1, FIX := 1, SIGNED := FALSE,	VAR_OUT:= MesDataExd.AX_STR[10].MesUdc);
	MW( WORD_STRONG:= MesBlock_Temp[4][ 75], SIZE := 1, FIX := 2, SIGNED := FALSE,	VAR_OUT:= MesDataExd.AX_STR[10].MesPdc);
	MW( WORD_STRONG:= MesBlock_Temp[4][ 93], SIZE := 1, FIX := 1, SIGNED := FALSE,	VAR_OUT:= MesDataExd.AX_STR[11].MesIdc);
	MW( WORD_STRONG:= MesBlock_Temp[4][ 94], SIZE := 1, FIX := 1, SIGNED := FALSE,	VAR_OUT:= MesDataExd.AX_STR[11].MesUdc);
	MW( WORD_STRONG:= MesBlock_Temp[4][ 95], SIZE := 1, FIX := 2, SIGNED := FALSE,	VAR_OUT:= MesDataExd.AX_STR[11].MesPdc);
	MW( WORD_STRONG:= MesBlock_Temp[4][113], SIZE := 1, FIX := 1, SIGNED := FALSE,	VAR_OUT:= MesDataExd.AX_STR[12].MesIdc);
	MW( WORD_STRONG:= MesBlock_Temp[4][114], SIZE := 1, FIX := 1, SIGNED := FALSE,	VAR_OUT:= MesDataExd.AX_STR[12].MesUdc);
	MW( WORD_STRONG:= MesBlock_Temp[4][115], SIZE := 1, FIX := 2, SIGNED := FALSE,	VAR_OUT:= MesDataExd.AX_STR[12].MesPdc);
	
	MesDataExd.MesData.MesU := (MesDataExd.MesU12 + MesDataExd.MesU23 +MesDataExd.MesU31)/3;

END_IF
END_METHOD

METHOD M_StartStop 
VAR_INPUT
END_VAR
VAR
	KK : UINT;
	AX_ADR_MB			: WORD := 40009;
	AX_QTY_MB			: ARRAY[1..2] OF BYTE := [2, 2];
	MotStart			: WORD := 569;
	MotStop				: WORD := 381;
	
END_VAR
SUPER^.M_StartStop() ;

Trig_CmdP(CLK := CmdP_IO);
Trig_CmdQ(CLK := CmdQ_IO);
Trig_CmdPF(CLK := CmdPF_IO);


MesDataExd.CmdStart_Ack := RS_StartStop.Q1;

IF IN_CmdStart THEN
	IN_CmdStart := FALSE;
END_IF

IF IN_CmdStop THEN
	IN_CmdStop := FALSE;
END_IF

IF Trig_CmdQ.Q THEN
	CmdQ_IO := FALSE;
	MesDataExd.CmdQ_Ack := TRUE;
	MesDataExd.CmdPF_Ack := FALSE;
END_IF

IF Trig_CmdPF.Q THEN
	CmdPF_IO := FALSE;
	MesDataExd.CmdQ_Ack := FALSE;
	MesDataExd.CmdPF_Ack := TRUE;
END_IF

IF Trig_CmdP.Q THEN
	CmdP_IO := FALSE;
	MesDataExd.CmdP_Ack := NOT MesDataExd.CmdP_Ack;
END_IF
END_METHOD

METHOD M_StateManager
//////////////////
// Detect which is the state of the inverter. IF loss of communication MesState =0 , the last inverter state is kept .  
/////////////////

VAR 
	// Method local variables (reinitialized at each cycle) 

	
END_VAR
//O=Stopped, 1 = MPPT, 2 = Sleeping, 3 = Starting, 4 = Throttled, 5 = Shutting down, 6 = Fault, 7 = Standby
MesDataExd.MesData.MesState := 0;

IF MesDataExd.MesData.MesState_Inv =1 THEN
	MesDataExd.MesData.MesState.0 			:= 1  ;
	
ELSIF  MesDataExd.MesData.MesState_Inv = 2 THEN
	MesDataExd.MesData.MesState.4 			:= 1  ;
	
ELSIF  MesDataExd.MesData.MesState_Inv = 3 THEN
	MesDataExd.MesData.MesState.3 			:= 1  ;
	
ELSIF  MesDataExd.MesData.MesState_Inv = 4 THEN
	MesDataExd.MesData.MesState.1 			:= 1  ;
	
ELSIF  MesDataExd.MesData.MesState_Inv = 5 THEN
	MesDataExd.MesData.MesState.4 			:= 1  ;
	
ELSIF  MesDataExd.MesData.MesState_Inv = 6 THEN
	MesDataExd.MesData.MesState.5 			:= 1  ;

ELSIF  MesDataExd.MesData.MesState_Inv = 7 THEN
	MesDataExd.MesData.MesState.6 			:= 1  ;
	
ELSIF  MesDataExd.MesData.MesState_Inv = 8 THEN
	MesDataExd.MesData.MesState.7 			:= 1  ;
	
END_IF



SUPER^.M_StateManager() ;
END_METHOD

END_FUNCTION_BLOCK

// ---- 01_Equipement_Library/Inverter/FB_SKID_PE_HEMG3.TcPOU
FUNCTION_BLOCK FB_SKID_PE_HEMG3

VAR_INPUT PERSISTENT
		ParamTcpPort				: UINT	:= 502;					  (* (NA) TCP port *)
		ParamIPAddress				: STRING; 						  (* (NA) Config: IP Adress of PV Inverter *)
		ParamID_SKID				: UINT;
		// Parameters of the Object (instance/model specific) 
		ParamTempoComAlarm				: TIME := T#30S ; 			  (* (s) Config : Tempo to detect LOC Alarm*)
		{attribute 'OPC.UA.DA' := '1'}
		ParamClockReadTime 				: TIME := T#2S;	  		  (* (Time) Read Modbus Frequency  *)
		{attribute 'OPC.UA.DA' := '1'}
 		ParamTimeout					: TIME := T#5S;			      (* (Time) Timeout for modbus reading *)
END_VAR

VAR_INPUT 
		
		IN_CmdToggleRead			: BOOL ;            		
		IN_CmdToggleWrite			: BOOL ; 
		IN_CmdReset_L				: BOOL ;
		
		MesDataExd					: SKID_PE_HEMG3; 					   // (NA) Inverter Object 
END_VAR

VAR	
	// M_READ VARIABLES//
		Trig_Cmd_Read				: R_TRIG; 
		Trig_Cmd_Write				: R_TRIG; 
                           
		
		ModbusRead	          		: FB_ModbusReadInputRegs; // (NA) FB for Modbus Reading
		AX_ModbusReadAlarm			: BOOL;
		AX_ModbusReadAlarmId		: UDINT;		
		AX_ModbusWriteAlarm			: BOOL;
		AX_ModbusWriteAlarmId		: UDINT;	
	
		MesBlock_Temp_1 			: ARRAY[1..5] OF WORD; 			// (NA) Temporary Block with multiple modbus reading 
		
	
	// M_ALARMMNGMT VARIABLES //
		TON_ComAlarm				: TON ; 						// Tempo before deteting loss of communication 
	    TON_ComWarning				: TON ;		 					// Tempo before detecting loss of communication                                                	
            
		MesWarningCom				: BOOL; 						// (NA) [P,H]  True if bad communication
		
		
	//M_EXECUTE VARIABLES //        	                        	
		TP1							: TP; 							// (NA) Tempo to define Modbus Reading Frequency 
		TP2 						: TP;	 						// (NA) Tempo to define Modbus Writing Frequency
		                            	                    		
		ClockRead					: BOOL;							// (NA) Modbus reading Clock
		ClockWrite 					: BOOL;							// (NA) Modbus writing Clock 		
		
		MesCP_Read			: BOOL := FALSE;	(* (NA) Cal : Permanent Condition for Read			  *)
		MesCP_Write			: BOOL := FALSE;	(* (NA) Cal : Permanenent Condition for Write		  *)
		
		
		
		
		bInit						: BOOL := TRUE;					// (NA) FB initialisation
END_VAR

METHOD M_AlarmManagement
//////////////////
// Manages IntelliGen Alarms
/////////////////

VAR 
	// Method local variables (reinitialized at each cycle) 
	FB_AlarmCodeManager : FB_AlarmCodeManager ; 
	KK				: BYTE;		// For Loop 
	bComError		: BOOL := TRUE;
	bComWarning 	: BOOL;

	AX_BJHS			: ARRAY[1..10] OF BOOL;
END_VAR
FOR KK := 1 TO 1 DO
	bComError := bCOmError AND AX_ModbusReadAlarm;
	bComWarning := bComWarning OR AX_ModbusReadAlarm;
END_FOR

TON_ComAlarm(IN := bComError, 		PT := T#30S, Q=> MesDataExd.MesAlarmCom);
TON_ComWarning(IN := bComWarning, 	PT := T#30S, Q=> MesWarningCom);

// ALARM CODE //
	FB_AlarmCodeManager(
		bAlarm1			:= MesDataExd.MesAlarmCom, 								// No communication frames for the past 30 seconds 					 			#COM
		bAlarm2			:= FALSE,												// 	
		bAlarm3			:= FALSE,												//  
		bAlarm4			:= FALSE,												// 	
		bAlarm5			:= FALSE,												// 
		bAlarm6			:= FALSE,												// 
		bAlarm7			:= FALSE,												//	
		bAlarm8			:= FALSE,												// 
		bAlarm9			:= FALSE,												// 
		bAlarm10		:= FALSE,												//  
		bAlarm11		:= FALSE,												// 		
		bAlarm12		:= FALSE,												//  
		bAlarm13		:= FALSE,												// 
		bAlarm14		:= FALSE,												// 
		bAlarm15		:= FALSE,												//
		wAlarmCode		=> MesDataExd.MesAlarmCode);					

// WARNING CODE //
	FB_AlarmCodeManager(
 		bAlarm1			:= MesWarningCom, 										// A frame failed for the last 30s 												#COM
		bAlarm2			:= FALSE,												//
		bAlarm3			:= NOT MesDataExd.MesCP_Read, 	  						// No permission to read from SCADA
		bAlarm4			:= FALSE,												//
		bAlarm5			:= NOT MesDataExd.MesCP_Write,							// No permission to write from SCADA							
		bAlarm6			:= FALSE,												//
		bAlarm7			:= FALSE,												// 
		bAlarm8			:= FALSE,												//
		bAlarm9			:= FALSE,												// 
		bAlarm10		:= FALSE,       										// 
		bAlarm11		:= FALSE,						 						// 
		bAlarm12		:= FALSE, 												//
		bAlarm13		:= FALSE,												// 
		bAlarm14		:= FALSE,												// 
		bAlarm15		:= FALSE, 												//
		wAlarmCode		=> MesDataExd.MesWarningCode);	

// EVENT CODE //
	FB_AlarmCodeManager(
		bAlarm1			:= FALSE,                            					//
		bAlarm2			:= FALSE,                                               //
		bAlarm3			:= FALSE,                                               //
		bAlarm4			:= FALSE,                                               //
		bAlarm5			:= FALSE,                                               //
		bAlarm6			:= FALSE,                                               //
		bAlarm7			:= FALSE,                                               //
		bAlarm8			:= FALSE,                                               //
		bAlarm9			:= FALSE,                                               //
		bAlarm10		:= FALSE,                                               //
		bAlarm11		:= FALSE, 												// 
		bAlarm12		:= FALSE,  												// 
		bAlarm13		:= FALSE, 												// 
		bAlarm14		:= FALSE, 												// 
		bAlarm15		:= FALSE,												// 		
		wAlarmCode		=>  MesDataExd.MesEventCode);
END_METHOD

METHOD M_CP
//////////////////
//  Emulator
/////////////////

VAR 
	// Method local variables (reinitialized at each cycle) 
	
END_VAR


SUPER^.M_CP() ; 




Trig_Cmd_Read(CLK:=IN_CmdToggleRead);
Trig_Cmd_Write(CLK:=IN_CmdToggleWrite);
	
IF Trig_Cmd_Read.Q THEN
	IN_CmdToggleRead := FALSE;
	MesDataExd.MesCP_Read := NOT MesDataExd.MesCP_Read;
END_IF


IF Trig_Cmd_Write.Q THEN
	IN_CmdToggleWrite := FALSE;
	MesDataExd.MesCP_Write := NOT MesDataExd.MesCP_Write;
END_IF
END_METHOD

METHOD M_Execute
//////////////////
//  Method Calls 
/////////////////

VAR 
	// Method local variables (reinitialized at each cycle) 

END_VAR
IF  bInit THEN
	M_Init();
	bInit:= FALSE ; 
ELSIF CmdInit_G THEN 
	bInit:= TRUE ;
END_IF

// READING AND WRITING CLOCK //
	TP1(IN:=NOT TP1.Q , PT:= ParamClockReadTime);
	ClockRead 				:= TP1.Q;
	

// PERMANENT CONDITIONS //	
	M_CP() ; 
	
// METHODS CALLS//
	M_Read();
	
//M_Evaluate();
	M_AlarmManagement();
END_METHOD

METHOD M_Init
VAR_INPUT
END_VAR
END_METHOD

{attribute 'object_name' := 'M_Read'}
METHOD M_Read
//////////
// Read Method for PE SKID HEMK : Modbus reading
//////////
VAR
	// Method local variables (reinitialized at each cycle) 
	
	AX_QTY_MB			: ARRAY[1..1] OF WORD := [5];
	AX_ADR_MB			: ARRAY[1..1] OF WORD := [0]; 	
	
	EacInj_Interm1		: ULINT;
	EacCon_Interm1		: ULINT;
	EreacCapa_Interm1	: ULINT;
	EreacInd_Interm1	: ULINT;
	EacInj_Day_Interm1	: ULINT;
	
	EacInj_Interm2		: ULINT;
	EacCon_Interm2		: ULINT;
	EreacCapa_Interm2	: ULINT;
	EreacInd_Interm2	: ULINT;
	EacInj_Day_Interm2	: ULINT;
	
	Temp_Cells_Transfo	: WORD;
	Temp_Cells_Transfo_2: WORD;
	Temp_Cells_Transfo_3: WORD;
	Temp_Cells_Transfo_4: WORD;
	
	KK					: BYTE;						 // Index to loop over modbus blocks 	
	JJ					: BYTE;
END_VAR
// CP-Read / Write 

IF  MesDataExd.MesCP_Read THEN		

// MODBUS REQUEST//
	//String Measurements
	ModbusRead
	(
		nTCPPort		:= ParamTcpPort,
		ClockRead		:= MesDataExd.MesCP_Read AND ClockRead, 
		Reset			:= CmdClearFault_G OR IN_CmdReset_L,
		sIPAddr			:= ParamIPAddress , 
		nUnitID			:= 1, 
		tTimeout		:= ParamClockReadTime,
		nQuantity		:= 5, 
		nMBAddr			:= 0, 
		cbLength		:= SIZEOF(MesBlock_Temp_1), 
		pDestAddr		:= ADR(MesBlock_Temp_1), 
		ErrorId			=> AX_ModbusReadAlarmId,
		ModbusReadAlarm => AX_ModbusReadAlarm
	);	
	// Cells and transformers 
	
		MesDataExd.MesDisparoTemp_Transformador1				:= MesBlock_Temp_1[1].0;                            	
		MesDataExd.MesAlarmTemp_Transformador1					:= MesBlock_Temp_1[1].1;                            	
		MesDataExd.MesDisparoPresion_Transformador1				:= MesBlock_Temp_1[1].2;                            	
		MesDataExd.MesDisparoOil_Transformador1					:= MesBlock_Temp_1[1].3;                            	
		MesDataExd.MesSeccionador1_Abierto						:= MesBlock_Temp_1[1].4;                            	
		MesDataExd.MesEarth1_Abierto							:= MesBlock_Temp_1[1].6;                            	
		MesDataExd.MesMonitorGas								:= MesBlock_Temp_1[1].7;                            	
		MesDataExd.MesSeccionador2_Abierto						:= MesBlock_Temp_1[1].8;                            	
		MesDataExd.MesEarth2_Abierto							:= MesBlock_Temp_1[1].10;                               	
		MesDataExd.MesSeccionadorMain1_Abierto					:= MesBlock_Temp_1[1].11;                            	
		MesDataExd.MesEarthMain1_Abierto						:= MesBlock_Temp_1[1].13;                          	
		MesDataExd.MesCb1_Abierto								:= MesBlock_Temp_1[1].14;   
		MesDataExd.MesProtectRelay1_fallo						:= MesBlock_Temp_1[2].0;
		MesDataExd.MesProtectRelay1_overvoltage					:= MesBlock_Temp_1[2].1;
		MesDataExd.MesProtectRelay1_springloaded				:= MesBlock_Temp_1[2].2;
		MesDataExd.MesMonitorGas2								:= MesBlock_Temp_1[2].3;
    
		MesDataExd.MesDisparoTemp_Transformador2				:= MesBlock_Temp_1[2].13;
		MesDataExd.MesAlarmTemp_Transformador2					:= MesBlock_Temp_1[2].14;
		MesDataExd.MesDisparoPresion_Transformador2				:= MesBlock_Temp_1[2].15;
		MesDataExd.MesDisparoOil_Transformador2					:= MesBlock_Temp_1[3].0;                             	
		MesDataExd.MesSeccionadorMain2_Abierto					:= MesBlock_Temp_1[3].1;   
		MesDataExd.MesEarth2_Abierto							:= MesBlock_Temp_1[3].3;  
		MesDataExd.MesCb2_Abierto								:= MesBlock_Temp_1[3].4;  
		MesDataExd.MesProtectRelay2_fallo						:= MesBlock_Temp_1[3].6;
		MesDataExd.MesProtectRelay2_overvoltage					:= MesBlock_Temp_1[3].6;
		MesDataExd.MesProtectRelay2_springloaded				:= MesBlock_Temp_1[3].8;
		IF ParamID_SKID = 2 OR ParamID_SKID = 3 THEN
			MesDataExd.MesTemp1									:= WORD_TO_REAL(MesBlock_Temp_1[3])/10;
		ELSE
			MesDataExd.MesTemp1									:= WORD_TO_REAL(MesBlock_Temp_1[4])/10;	
			MesDataExd.MesTemp2									:= WORD_TO_REAL(MesBlock_Temp_1[5])/10;
		END_IF

END_IF
END_METHOD

END_FUNCTION_BLOCK

// ---- 01_Equipement_Library/IPC/FB_IPC.TcPOU
FUNCTION_BLOCK FB_IPC

VAR_INPUT PERSISTENT 
	ParamTempoRestart		: TIME 	:= T#30S ;	(* (s)Tempo to wait before resupplying the IPC *)	
END_VAR
      	
VAR_INPUT  
	MesDataExd				: IPC_Standard;
	Heure_Local     		: TIMESTRUCT;
	IN_CmdRestart 			: BOOL;	
	IN_CmdReset_L			: BOOL;			// (NA) External Reset Command
END_VAR     

VAR_OUTPUT
	//Child objects
	OUT_CmdOpen_IO			: BOOL;	
END_VAR        	
      	
VAR                 	
	bInit					: BOOL := TRUE;	// Booleen d'initialisation		
	TP_Restart				: TP;
	// State Mananger //
	MesState				: BYTE; 		// Cal  : state
END_VAR

METHOD M_AlarmManagement
//////////////////
// Generates object alarms and manages resets. 
//////////////////

VAR 
	// Method local variables (reinitialized at each cycle) 
	FB_AlarmCodeManager		: FB_AlarmCodeManager ;  
END_VAR
	
// ALARM CODE //
	FB_AlarmCodeManager(
		bAlarm1				:= FALSE,						//
		bAlarm2				:= FALSE,                       //
		bAlarm3				:= FALSE,                       //
		bAlarm4				:= FALSE,                       //
		bAlarm5				:= FALSE,                       //
		bAlarm6				:= FALSE,                       //
		bAlarm7				:= FALSE,                       //
		bAlarm8				:= FALSE,                       //
		bAlarm9				:= FALSE,                       //
		bAlarm10			:= FALSE,                       //
		bAlarm11			:= FALSE,                       //
		bAlarm12			:= FALSE,						//
		bAlarm13			:= FALSE ,                      //
		bAlarm14			:= FALSE ,                      //
		bAlarm15			:= FALSE,                       //
		wAlarmCode			=>MesDataExd.MesData.MesAlarmCode);       
			                                                
// WARNING CODE //                                          
	FB_AlarmCodeManager(
		bAlarm1				:= FALSE, 						//				
		bAlarm2				:= FALSE,                       //
		bAlarm3				:= FALSE,                       //
		bAlarm4				:= FALSE,                       //
		bAlarm5				:= FALSE,                       //
		bAlarm6				:= FALSE,                       //
		bAlarm7				:= FALSE,                       //
		bAlarm8				:= FALSE,                       //
		bAlarm9				:= FALSE,                       //
		bAlarm10			:= FALSE,                       //
		bAlarm11			:= FALSE,                       //
		bAlarm12			:= FALSE,                       //
		bAlarm13			:= FALSE,                       //
		bAlarm14			:= FALSE,                       //
		bAlarm15			:= FALSE,                       //
		wAlarmCode			=>MesDataExd.MesData.MesWarningCode);
		
// EVENT CODE //
	FB_AlarmCodeManager(
		bAlarm1			:= OUT_CmdOpen_IO, 					// Open command
		bAlarm2			:= FALSE , 							//
		bAlarm3			:= FALSE,                           //
		bAlarm4			:= FALSE,                           //
		bAlarm5			:= FALSE,                           //
		bAlarm6			:= FALSE,                           //
		bAlarm7			:= FALSE,                           //
		bAlarm8			:= FALSE,                           //
		bAlarm9			:= FALSE,                           //
		bAlarm10		:= FALSE,                           //
		bAlarm11		:= FALSE,                           //
		bAlarm12		:= FALSE,                           //
		bAlarm13		:= FALSE,                           //
		bAlarm14		:= FALSE,                           //
		bAlarm15		:= FALSE,                           //
		wAlarmCode		=>MesDataExd.MesData.MesEventCode);
END_METHOD

METHOD M_Execute : BOOL
VAR_INPUT
END_VAR
IF bInit THEN
	M_Init();
ELSIF CmdInit_G OR IN_CmdReset_L THEN
	bInit := TRUE;
ELSE
	M_OpenClose(); 
	M_StateManager();
END_IF
END_METHOD

METHOD M_Init : BOOL
VAR_INPUT
END_VAR
bInit := FALSE;
END_METHOD

METHOD M_OpenClose
//////////////////
// Manages restart of the IPC 
//////////////////

VAR 
	// Method local variables (reinitialized at each cycle) 
	
END_VAR

// Rest Command
TP_Restart(IN:= IN_CmdRestart , PT:=ParamTempoRestart) ;
OUT_CmdOpen_IO := TP_Restart.Q ;  // Impulsion that goes back to zero as soon as the state of the TP goes down 

IF  IN_CmdRestart THEN
	 IN_CmdRestart := FALSE;
END_IF
END_METHOD

METHOD M_StateManager
//////////////////
// IPC off -> State.2 = 1, IPC on -> State.0 = 1 
/////////////////

VAR 
	// Method local variables (reinitialized at each cycle) 
	
END_VAR
// OPERATIONNAL INDEX //
IF NOT  OUT_CmdOpen_IO THEN 
	MesState.2 := 1;
ELSE
	MesState.0 := 1;
END_IF
END_METHOD

END_FUNCTION_BLOCK

// ---- 01_Equipement_Library/Operation Meter/FB_PM_ION9200.TcPOU
FUNCTION_BLOCK FB_PM_ION9200 EXTENDS FB_PM_Base
//////////////////
// Measurement Solution based on Digiware, but access through PMS Socomec
//////////////////
VAR CONSTANT
	// Characteristics of the object (Same for all instances)
			
END_VAR

VAR_INPUT PERSISTENT
	// Parameters of the Object (instance specific) 
	{attribute 'OPC.UA.DA' := '1'} 
	ParamUnitID					: BYTE 		:= 1 ;								(* (NA) Unit ID*)
//	ParamInInterfaceSub			: BOOL 		:= TRUE; 							// (NA) Serial interface RS422/RS485 TYPE (0:EL6021,1:SUB9)
	{attribute 'OPC.UA.DA' := '1'} 
	ParamIPAddress		   		: STRING 	:= '192.168.20.15'; 				(* (NA) IP Adress of ION7650 *)
	{attribute 'OPC.UA.DA' := '1'} 
	ParamTcpPort				: UINT 		:= 502;								(* (NA) TCP port			*)

END_VAR

VAR_OUTPUT
	//Child objects
	
END_VAR

VAR_INPUT 
			MesDataExd				: PM_ION9200;								// (NA) Structure of the PM3250
END_VAR


VAR                                                  								                                          								
	//M_READ VARIABLES//
		ModbusRead					: ARRAY[1..4] OF FB_ModbusRead;
		AX_Quantity					: ARRAY[1..4] OF WORD	:= [1,  	16, 	112,		8];					// (NA) Quantity of blocks to read
		AX_Address					: ARRAY[1..4] OF WORD	:= [1841,	2699, 	2999,	3143];					// (NA) Start address of the read
		MesBlock_Temp 				: ARRAY[1..4] OF ARRAY[1..125] OF WORD;	// (NA) Temporary Block with multiple modbus reading (U30 + I35)	
		OutErrorMbRead				: ARRAY[1..4] OF BOOL;
		OutErrorMbReadId			: ARRAY[1..4] OF UDINT;
		
		RTrigI						: R_TRIG;
	//M_INIT VARIABLES //
		OutFBCompleteted			: BOOL;
	// ION was reset to 0 
		IONCount_PossibleReset		: BOOL := TRUE; 						// (NA) The active power of the PM ION7650 is between 1000 and  10m 
		

	bTestComError : BOOL;
		
END_VAR

METHOD M_AlarmManagement
//////////////////
// Digiware measurement tool alarm and warning management
/////////////////

VAR 
	// Method local variables (reinitialized at each cycle) 
	FB_AlarmCodeManager			: FB_AlarmCodeManager ; 
	
	KK							: BYTE ;		// For loop
	
	CMWarning					: BOOL;			// At least one Digiware device in Alarm
	CMAlarm						: BOOL;			// At least one Digiware device in Alarm
	
END_VAR
TON_ComAlarm(IN:= (OutErrorMbRead[1] AND OutErrorMbRead[2] AND OutErrorMbRead[3]) or bTestComError , PT:= ParamTempoComAlarm, Q=>MesDataExd.MesData.MesAlarmCom) ;	

//					General com alarm : All the read FB fucked up

// ALARM CODE //
	FB_AlarmCodeManager( 
		bAlarm1			:=MesDataExd.MesData.MesAlarmCom, 					// Communication Error  #COM
		bAlarm2			:=FALSE, 									// 
		bAlarm3			:=FALSE, 									// 
		bAlarm4			:=FALSE, 									// 
		bAlarm5			:=FALSE, 									//
		bAlarm6			:=FALSE, 									//
		bAlarm7			:=FALSE, 									//
		bAlarm8			:=FALSE, 									//
		bAlarm9			:=FALSE, 									//
		bAlarm10		:=FALSE, 									//
		bAlarm11		:=FALSE, 									//
		bAlarm12		:=FALSE, 									//
		bAlarm13		:=FALSE, 									//
		bAlarm14		:=FALSE, 									//
		bAlarm15		:= FALSE , 									//						 
		wAlarmCode		=>MesDataExd.MesData.MesAlarmCode);

// WARNING CODE //
	FB_AlarmCodeManager(		
		bAlarm1			:=	MesWarningCom,				 			// Communication Warning #COM	
		bAlarm2			:=FALSE, 									// 
		bAlarm3			:=FALSE, 									// 
		bAlarm4			:=FALSE, 									// 
		bAlarm5			:=FALSE, 									//
		bAlarm6			:=FALSE, 									//
		bAlarm7			:=FALSE, 									//
		bAlarm8			:=FALSE, 									//
		bAlarm9			:=FALSE, 									//
		bAlarm10		:=FALSE, 									//
		bAlarm11		:=FALSE, 									//
		bAlarm12		:=FALSE, 									//
		bAlarm13		:=FALSE, 									//
		bAlarm14		:=FALSE, 									//
		bAlarm15		:=FALSE, 									//
		wAlarmCode		=>MesDataExd.MesData.MesWarningCode);
END_METHOD

METHOD M_CP
//////////////////
//  Emulator
/////////////////

VAR 
	// Method local variables (reinitialized at each cycle) 
	
END_VAR


SUPER^.M_CP() ; 




Trig_Cmd_Read(CLK:=IN_CmdToggleRead);
	
IF Trig_Cmd_Read.Q THEN
	IN_CmdToggleRead := FALSE;
	MesDataExd.MesData.MesCP_Read := NOT MesDataExd.MesData.MesCP_Read;
END_IF
END_METHOD

METHOD M_Evaluate : BOOL
VAR_INPUT
END_VAR
END_METHOD

METHOD M_Init
VAR 

END_VAR
(*FB_ModbusRead(InTimeout:= ParamTimeout,
				 InUnitID:= DINT_TO_BYTE(ParamUnitID),
				 InQuantity:= 125,	
				 InInterfaceSub:= ParamInInterfaceSub,
				 InFunctionRead := FALSE);
*)
	
AX_Quantity[1] := 125;
AX_Address[1]  := 149;

ParamClockReadTime := T#200ms;
END_METHOD

METHOD M_Read
//////////////////
//  Read Modbus Variable for ION7650. 
/////////////////
VAR 
	// Method local variables (reinitialized at each cycle) 
	MW 					: FB_MergeWordsToDint; 
	MW_Real				: FB_MergeWordsToFloat; 
	KK					: BYTE;  						// FOR Loop 

	NbRead: UDINT;
END_VAR
IF MesDataExd.MesData.MesCP_Read THEN
	ModbusRead[1](
		pDestAddr 			:= ADR(MesBlock_Temp[1]),
		sIPAddr 			:= ParamIPAddress,
		tTimeout 			:= ParamClockReadTime,
		nTcpPort 			:= ParamTcpPort,
		nQuantity			:= AX_Quantity[1],
		nMBAddr				:= AX_Address[1],
		cbLength			:= SIZEOF(MesBlock_Temp[1]),
		nUnitID				:= 100,
		ClockRead			:= ClockRead,
		OUT_NbRead			=> NbRead,
		ModbusReadAlarm		=> OutErrorMbRead[1],
		ErrorId				=> OutErrorMbReadId[1]
	);
	
	ModbusRead[2](
		pDestAddr 			:= ADR(MesBlock_Temp[2]),
		sIPAddr 			:= ParamIPAddress,
		tTimeout 			:= ParamClockReadTime,
		nTcpPort 			:= ParamTcpPort,
		nQuantity			:= AX_Quantity[2],
		nMBAddr				:= AX_Address[2],
		cbLength			:= SIZEOF(MesBlock_Temp[2]),
		nUnitID				:= 100,
		ClockRead			:= ClockRead,
		OUT_NbRead			=> NbRead,
		ModbusReadAlarm		=> OutErrorMbRead[2],
		ErrorId				=> OutErrorMbReadId[2]
	);
	
	ModbusRead[3](
		pDestAddr 			:= ADR(MesBlock_Temp[3]),
		sIPAddr 			:= ParamIPAddress,
		tTimeout 			:= ParamClockReadTime,
		nTcpPort 			:= ParamTcpPort,
		nQuantity			:= AX_Quantity[3],
		nMBAddr				:= AX_Address[3],
		cbLength			:= SIZEOF(MesBlock_Temp[3]),
		nUnitID				:= 100,
		ClockRead			:= ClockRead,
		OUT_NbRead			=> NbRead,
		ModbusReadAlarm		=> OutErrorMbRead[3],
		ErrorId				=> OutErrorMbReadId[3]
	);

	ModbusRead[4](
		pDestAddr 			:= ADR(MesBlock_Temp[4]),
		sIPAddr 			:= ParamIPAddress,
		tTimeout 			:= ParamClockReadTime,
		nTcpPort 			:= ParamTcpPort,
		nQuantity			:= AX_Quantity[4],
		nMBAddr				:= AX_Address[4],
		cbLength			:= SIZEOF(MesBlock_Temp[4]),
		nUnitID				:= 100,
		ClockRead			:= ClockRead,
		OUT_NbRead			=> NbRead,
		ModbusReadAlarm		=> OutErrorMbRead[4],
		ErrorId				=> OutErrorMbReadId[4]
	);	
		

	// Block 1
		MesDataExd.MesSeconds := WORD_TO_UINT(MesBlock_Temp[1][1]);
		
	// Block 2
		MW_Real(WORD_STRONG:= MesBlock_Temp[2][1], WORD_WEAK:= MesBlock_Temp[2][2], var_out := MesDataExd.MesData.MesEActProd);
		MW_Real(WORD_STRONG:= MesBlock_Temp[2][3], WORD_WEAK:= MesBlock_Temp[2][4], var_out := MesDataExd.MesData.MesEActCons);
	
	// Block 3	
		MW_Real(WORD_STRONG:= MesBlock_Temp[3][  1], WORD_WEAK:= MesBlock_Temp[3][  2], var_out := MesDataExd.MesData.MesI1);
		MW_Real(WORD_STRONG:= MesBlock_Temp[3][  3], WORD_WEAK:= MesBlock_Temp[3][  4], var_out := MesDataExd.MesData.MesI2);
		MW_Real(WORD_STRONG:= MesBlock_Temp[3][  5], WORD_WEAK:= MesBlock_Temp[3][  6], var_out := MesDataExd.MesData.MesI3);
		MW_Real(WORD_STRONG:= MesBlock_Temp[3][ 11], WORD_WEAK:= MesBlock_Temp[3][ 12], var_out := MesDataExd.MesData.MesI);
		MW_Real(WORD_STRONG:= MesBlock_Temp[3][ 21], WORD_WEAK:= MesBlock_Temp[3][ 22], var_out := MesDataExd.MesData.MesU12);
		MW_Real(WORD_STRONG:= MesBlock_Temp[3][ 23], WORD_WEAK:= MesBlock_Temp[3][ 24], var_out := MesDataExd.MesData.MesU23);
		MW_Real(WORD_STRONG:= MesBlock_Temp[3][ 25], WORD_WEAK:= MesBlock_Temp[3][ 26], var_out := MesDataExd.MesData.MesU31);
		MW_Real(WORD_STRONG:= MesBlock_Temp[3][ 27], WORD_WEAK:= MesBlock_Temp[3][ 28], var_out := MesDataExd.MesData.MesU);
		MW_Real(WORD_STRONG:= MesBlock_Temp[3][ 29], WORD_WEAK:= MesBlock_Temp[3][ 30], var_out := MesDataExd.MesData.MesV1);
		MW_Real(WORD_STRONG:= MesBlock_Temp[3][ 31], WORD_WEAK:= MesBlock_Temp[3][ 32], var_out := MesDataExd.MesData.MesV2);
		MW_Real(WORD_STRONG:= MesBlock_Temp[3][ 33], WORD_WEAK:= MesBlock_Temp[3][ 34], var_out := MesDataExd.MesData.MesV3);
		MW_Real(WORD_STRONG:= MesBlock_Temp[3][ 37], WORD_WEAK:= MesBlock_Temp[3][ 38], var_out := MesDataExd.MesData.MesV);
		MW_Real(WORD_STRONG:= MesBlock_Temp[3][ 55], WORD_WEAK:= MesBlock_Temp[3][ 56], var_out := MesDataExd.MesData.MesP1);
		MW_Real(WORD_STRONG:= MesBlock_Temp[3][ 57], WORD_WEAK:= MesBlock_Temp[3][ 58], var_out := MesDataExd.MesData.MesP2);
		MW_Real(WORD_STRONG:= MesBlock_Temp[3][ 59], WORD_WEAK:= MesBlock_Temp[3][ 60], var_out := MesDataExd.MesData.MesP3);
		MW_Real(WORD_STRONG:= MesBlock_Temp[3][ 61], WORD_WEAK:= MesBlock_Temp[3][ 62], var_out := MesDataExd.MesData.MesP);
		MW_Real(WORD_STRONG:= MesBlock_Temp[3][ 63], WORD_WEAK:= MesBlock_Temp[3][ 64], var_out := MesDataExd.MesData.MesQ1);
		MW_Real(WORD_STRONG:= MesBlock_Temp[3][ 65], WORD_WEAK:= MesBlock_Temp[3][ 66], var_out := MesDataExd.MesData.MesQ2);
		MW_Real(WORD_STRONG:= MesBlock_Temp[3][ 67], WORD_WEAK:= MesBlock_Temp[3][ 68], var_out := MesDataExd.MesData.MesQ3);
		MW_Real(WORD_STRONG:= MesBlock_Temp[3][ 69], WORD_WEAK:= MesBlock_Temp[3][ 70], var_out := MesDataExd.MesData.MesQ);
		MW_Real(WORD_STRONG:= MesBlock_Temp[3][ 71], WORD_WEAK:= MesBlock_Temp[3][ 72], var_out := MesDataExd.MesData.MesS1);
		MW_Real(WORD_STRONG:= MesBlock_Temp[3][ 73], WORD_WEAK:= MesBlock_Temp[3][ 74], var_out := MesDataExd.MesData.MesS2);
		MW_Real(WORD_STRONG:= MesBlock_Temp[3][ 75], WORD_WEAK:= MesBlock_Temp[3][ 76], var_out := MesDataExd.MesData.MesS3);
		MW_Real(WORD_STRONG:= MesBlock_Temp[3][ 77], WORD_WEAK:= MesBlock_Temp[3][ 78], var_out := MesDataExd.MesData.MesS);
		MW_Real(WORD_STRONG:= MesBlock_Temp[3][111], WORD_WEAK:= MesBlock_Temp[3][112], var_out := MesDataExd.MesData.MesFreq);

	// Block 4
		MW_Real(WORD_STRONG:= MesBlock_Temp[4][  1], WORD_WEAK:= MesBlock_Temp[4][  2], var_out := MesDataExd.MesData.MesCosPhi1);
		MW_Real(WORD_STRONG:= MesBlock_Temp[4][  3], WORD_WEAK:= MesBlock_Temp[4][  4], var_out := MesDataExd.MesData.MesCosPhi2);
		MW_Real(WORD_STRONG:= MesBlock_Temp[4][  5], WORD_WEAK:= MesBlock_Temp[4][  6], var_out := MesDataExd.MesData.MesCosPhi3);
		MW_Real(WORD_STRONG:= MesBlock_Temp[4][  7], WORD_WEAK:= MesBlock_Temp[4][  8], var_out := MesDataExd.MesData.MesCosPhi);


		MesDataExd.MesData.MesP1	:= - MesDataExd.MesData.MesP1 /1000;
		MesDataExd.MesData.MesP2    := - MesDataExd.MesData.MesP2 /1000;
		MesDataExd.MesData.MesP3    := - MesDataExd.MesData.MesP3 /1000;
		MesDataExd.MesData.MesP     := - MesDataExd.MesData.MesP  /1000;
		MesDataExd.MesData.MesQ1    := - MesDataExd.MesData.MesQ1 /1000;
		MesDataExd.MesData.MesQ2    := - MesDataExd.MesData.MesQ2 /1000;
		MesDataExd.MesData.MesQ3    := - MesDataExd.MesData.MesQ3 /1000;
		MesDataExd.MesData.MesQ     := - MesDataExd.MesData.MesQ  /1000;		
END_IF
END_METHOD

END_FUNCTION_BLOCK

// ---- 01_Equipement_Library/Operation Meter/FB_PM_Base.TcPOU
FUNCTION_BLOCK FB_PM_Base 
//////////////////
// Measurement Solution. Base FB
//////////////////
VAR_INPUT PERSISTENT
	// Parameters of the Object (instance specific) 
	ParamTempoComAlarm				: TIME 		:= T#10S ; 						(* (s) Config : Tempo to detect LOC Alarm*)
	{attribute 'OPC.UA.DA' := '1'} 
	ParamClockReadTime 				: TIME 		:= TIME#200MS;	  				(* (ms) Read Modbus period  *)
	ParamTimeout					: TIME  	:= T#2S ;			  			(* (s) Timeout for modbus reading*)
	
	
END_VAR

VAR_INPUT
	//Child objects
	IN_CmdToggleRead				: BOOL ; 
	IN_CmdReset_L					: BOOL ;									// (NA) External Reset Command

END_VAR
VAR
	//M_ALARMMANAGEMENT VARIABLES//
		TON_ComAlarm				: TON ; 									// Tempo before detecting loss of communication 
	    TON_ComWarning				: TON ; 									// Tempo before detecting loss of one frame                                               								
                                            								    
		MesWarningCom				: BOOL ; 									// True if bad communication 
                                                                                 
	//M_READ VARIABLES//                                                         
//	MesDataExd		AT %Q*	: PM ;                                 
		ClockRead			AT %Q*	: BOOL ;	 								// Clock Read
                                                                                
		                                                                         
	//M_INIT VARIABLES //
		bInit						: BOOL 				:= TRUE ; 							// (NA) Initialize object parameters at first cycle 
		                                                                         
	// M_EXECUTE VARIABLES //
		TP1							: TP ; 												// (NA) Tempo to define Modbus Reading Frequency  
                                                             	                                                                                                                                                      
		//MesCP_Read					: BOOL;													// (NA) Permanent conditions to activate method
        Trig_Cmd_Read				: R_TRIG;      

                 
END_VAR

METHOD M_AlarmManagement
//////////////////
// Digiware measurement tool alarm and warning management
/////////////////

VAR 
	
END_VAR
END_METHOD

METHOD M_CP
//////////////////
//  Emulator
/////////////////

VAR 
	// Method local variables (reinitialized at each cycle) 
	
END_VAR
END_METHOD

METHOD M_Execute
//////////////////
//  Method Calls 
/////////////////
VAR 
	// Method local variables (reinitialized at each cycle) 
	// EMULATOR

	
END_VAR
// READING AND WRITING CLOCK //
	TP1(IN:=NOT TP1.Q , PT:= ParamClockReadTime);
	ClockRead 		:= TP1.Q;

// PERMANENT CONDITIONS //
	M_CP() ; 
	
// METHODS CALLS //
	IF bInit THEN
		M_Init() ; 
		bInit					:= FALSE ; 
	ELSIF CmdInit_G OR IN_CmdReset_L THEN 
		bInit:= TRUE ;		
	END_IF

	M_Read() ; 
	M_AlarmManagement();
END_METHOD

METHOD M_Init
VAR 

END_VAR
END_METHOD

METHOD M_Read
//////////////////
//  Read Modbus Variable for PCS . 
/////////////////
VAR 
	// Method local variables (reinitialized at each cycle) 
	
END_VAR
END_METHOD

END_FUNCTION_BLOCK

// ---- 01_Equipement_Library/Operation Meter/FB_PM_PM5XXX.TcPOU
FUNCTION_BLOCK FB_PM_PM5XXX EXTENDS FB_PM_Base
//////////////////
// Schneider Power Meter PM5340. PM auxiliaries
//////////////////
VAR CONSTANT
	// Characteristics of the object (Same for all instances)
			
END_VAR

VAR_INPUT PERSISTENT
	// Parameters of the Object (instance specific) 
	ParamUnitID						: BYTE 	:= 1 ;				(* (NA) Unit ID   							*)	
	ParamTcpPort					: UINT	:= 502;				(* (NA) TCP port 							*)
	ParamIPAddress					: STRING;					(* (NA)	Config: IP Adress of PV INverter	*)
			
END_VAR

VAR_OUTPUT
	//Child objects
	
END_VAR

VAR_INPUT
	MesDataExd			AT %Q*		: PM_PM5XXX;
	IN_SwitchPos_IO					: BOOL; // Definition to be clarified during FAT
	
END_VAR

VAR
	// M_Read		
		FB_ModbusRead	          	: ARRAY[1..4] OF FB_ModbusRead;  // (NA) FB for Modbus Reading
		AX_ModbusReadAlarm			: ARRAY[1..4] OF BOOL;
		AX_ModbusReadAlarmId		: ARRAY[1..4] OF UDINT;		
	
		MesBlock_Temp_1 			: ARRAY [1..20]  OF WORD; 		// (NA) Temporary Block with multiple modbus reading 
		MesBlock_Temp_2 			: ARRAY [1..128] OF WORD; 		// (NA) Temporary Block with multiple modbus reading 
		MesBlock_Temp_3 			: ARRAY [1..128] OF WORD; 		// (NA) Temporary Block with multiple modbus reading 
		MesBlock_Temp_4 			: ARRAY [1..60]  OF WORD; 		// (NA) Temporary Block with multiple modbus reading 
		
		OutErrorMbRead				: ARRAY[1..5] OF BOOL;
		
		
		AX_QTY_MB			: ARRAY[1..4] OF WORD := [20, 112, 104, 60];
		AX_ADR_MB			: ARRAY[1..4] OF WORD := [2699, 2999, 13522, 21299]; 
END_VAR

METHOD M_AlarmManagement
//////////////////
//Alarms and warnings management
/////////////////

VAR 
	// Method local variables (reinitialized at each cycle) 
	FB_AlarmCodeManager			: FB_AlarmCodeManager; 
	
	KK							: BYTE;			// For loop
	
	CMWarning					: BOOL;			// At least one Digiware device in Alarm
	CMAlarm						: BOOL;			// At least one Digiware device in Alarm
	
END_VAR
	
TON_ComAlarm(IN:= OutErrorMbRead[1] AND OutErrorMbRead[2] AND OutErrorMbRead[3] AND OutErrorMbRead[4] AND OutErrorMbRead[5] , PT:= ParamTempoComAlarm, Q=> MesDataExd.MesData.MesAlarmCom);	
TON_ComWarning(IN:= OutErrorMbRead[1] OR OutErrorMbRead[2] OR OutErrorMbRead[3] OR OutErrorMbRead[4] OR OutErrorMbRead[5] , PT:= ParamTempoComAlarm, Q=>MesWarningCom);	

MesDataExd.MesAlarmSW_Open := NOT IN_SwitchPos_IO;  
// ALARM CODE //
	FB_AlarmCodeManager(
		bAlarm1			:= MesDataExd.MesData.MesAlarmCom, 			// Communication Error #COM
		bAlarm2			:= MesDataExd.MesAlarmSW_Open, 				// PM switch open
		bAlarm3			:=FALSE, 									// 
		bAlarm4			:=FALSE, 									// 
		bAlarm5			:=FALSE, 									//
		bAlarm6			:=FALSE, 									//
		bAlarm7			:=FALSE, 									//
		bAlarm8			:=FALSE, 									//
		bAlarm9			:=FALSE, 									//
		bAlarm10		:=FALSE, 									//
		bAlarm11		:=FALSE, 									//
		bAlarm12		:=FALSE, 									//
		bAlarm13		:=FALSE, 									//
		bAlarm14		:=FALSE, 									//
		bAlarm15		:= FALSE , 									// 							 
		wAlarmCode		=> MesDataExd.MesData.MesAlarmCode);

// WARNING CODE //
	FB_AlarmCodeManager(		
		bAlarm1			:=MesWarningCom	,				 			// Communication Warning #COM
		bAlarm2			:=FALSE, 						 			// 
		bAlarm3			:=FALSE, 						 			// 
		bAlarm4			:=FALSE, 						 			// 
		bAlarm5			:=FALSE, 						 			//
		bAlarm6			:=FALSE, 						 			//
		bAlarm7			:=FALSE, 						 			//
		bAlarm8			:=FALSE, 						 			//
		bAlarm9			:=FALSE, 						 			//
		bAlarm10		:=FALSE, 						 			//
		bAlarm11		:=FALSE, 						 			//
		bAlarm12		:=FALSE, 						 			//
		bAlarm13		:=FALSE, 						 			//
		bAlarm14		:=FALSE, 						 			//
		bAlarm15		:=FALSE, 						 			//
		wAlarmCode		=> MesDataExd.MesData.MesWarningCode);
END_METHOD

METHOD M_CP
//////////////////
//  Emulator
/////////////////

VAR 
	// Method local variables (reinitialized at each cycle) 
	
END_VAR


SUPER^.M_CP() ; 




Trig_Cmd_Read(CLK:=IN_CmdToggleRead);
	
IF Trig_Cmd_Read.Q THEN
	IN_CmdToggleRead := FALSE;
	MesDataExd.MesData.MesCP_Read := NOT MesDataExd.MesData.MesCP_Read;
END_IF
END_METHOD

METHOD M_Evaluate : BOOL
VAR_INPUT
END_VAR
END_METHOD

METHOD M_Init
VAR 

END_VAR
ParamClockReadTime := T#10s;
END_METHOD

METHOD M_Read
//////////////////
//  Read Modbus variables for Schneider PM models : PM5560, PM5563, PM5563RD. 
/////////////////
VAR 
	// Method local variables (reinitialized at each cycle) 
	MW_Float			: FB_MergeWordsToFloat;
	MW_UInt				: FB_MergeWordsToUint;
	
END_VAR

IF MesDataExd.MesData.MesCP_Read THEN	
	
		FB_ModbusRead[1]
	(
		nTCPPort		:= ParamTcpPort,
		ClockRead		:= MesDataExd.MesData.MesCP_Read AND ClockRead, 
		Reset			:= CmdClearFault_G OR IN_CmdReset_L,
		sIPAddr			:=ParamIPAddress,
		nUnitID			:= 255, 
		tTimeout		:= ParamTimeout,
		nQuantity		:= AX_QTY_MB[1], 
		nMBAddr			:= AX_ADR_MB[1], 
		cbLength		:= SIZEOF(MesBlock_Temp_1), 
		pDestAddr		:= ADR(MesBlock_Temp_1), 
		ModbusReadAlarm	=>AX_ModbusReadAlarm[1], 
		ErrorId			=> AX_ModbusReadAlarmId[1]
	);
	
	FB_ModbusRead[2]
	(
		nTCPPort		:= ParamTcpPort,
		ClockRead		:= MesDataExd.MesData.MesCP_Read AND ClockRead, 
		Reset			:= CmdClearFault_G OR IN_CmdReset_L,
		sIPAddr			:=ParamIPAddress, 
		nUnitID			:= 255, 
		tTimeout		:= ParamTimeout,
		nQuantity		:= AX_QTY_MB[2], 
		nMBAddr			:= AX_ADR_MB[2], 
		cbLength		:= SIZEOF(MesBlock_Temp_2), 
		pDestAddr		:= ADR(MesBlock_Temp_2), 
		ModbusReadAlarm	=>AX_ModbusReadAlarm[2], 
		ErrorId			=> AX_ModbusReadAlarmId[2]
	);
	
	FB_ModbusRead[3]
	(
		nTCPPort		:= ParamTcpPort,
		ClockRead		:= MesDataExd.MesData.MesCP_Read AND ClockRead, 
		Reset			:= CmdClearFault_G OR IN_CmdReset_L,
		sIPAddr			:=ParamIPAddress, 
		nUnitID			:= 255, 
		tTimeout		:= ParamTimeout,
		nQuantity		:= AX_QTY_MB[3], 
		nMBAddr			:= AX_ADR_MB[3], 
		cbLength		:= SIZEOF(MesBlock_Temp_3), 
		pDestAddr		:= ADR(MesBlock_Temp_3), 
		ModbusReadAlarm	=>AX_ModbusReadAlarm[3], 
		ErrorId			=> AX_ModbusReadAlarmId[3]
	);
	
	FB_ModbusRead[4]
	(
		nTCPPort		:= ParamTcpPort,
		ClockRead		:= MesDataExd.MesData.MesCP_Read AND ClockRead, 
		Reset			:= CmdClearFault_G OR IN_CmdReset_L,
		sIPAddr			:= ParamIPAddress , 
		nUnitID			:= 255, 
		tTimeout		:= ParamTimeout,
		nQuantity		:= AX_QTY_MB[4], 
		nMBAddr			:= AX_ADR_MB[4], 
		cbLength		:= SIZEOF(MesBlock_Temp_4), 
		pDestAddr		:= ADR(MesBlock_Temp_4), 
		ModbusReadAlarm	=> AX_ModbusReadAlarm[4], 
		ErrorId			=> AX_ModbusReadAlarmId[4]
	);
	
	MW_Float( WORD_STRONG := MesBlock_Temp_1[1],  WORD_WEAK := MesBlock_Temp_1[2],  VAR_OUT := MesDataExd.MesData.MesEActProd);
	MW_Float( WORD_STRONG := MesBlock_Temp_1[3],  WORD_WEAK := MesBlock_Temp_1[4],  VAR_OUT := MesDataExd.MesData.MesEActCons);
	MW_Float( WORD_STRONG := MesBlock_Temp_1[9],  WORD_WEAK := MesBlock_Temp_1[10], VAR_OUT := MesDataExd.MesData.MesEReactProd);
	MW_Float( WORD_STRONG := MesBlock_Temp_1[11], WORD_WEAK := MesBlock_Temp_1[12], VAR_OUT := MesDataExd.MesData.MesEReactCons);
	MW_Float( WORD_STRONG := MesBlock_Temp_1[17], WORD_WEAK := MesBlock_Temp_1[18], VAR_OUT := MesDataExd.MesEAppProd);
	MW_Float( WORD_STRONG := MesBlock_Temp_1[19], WORD_WEAK := MesBlock_Temp_1[20], VAR_OUT := MesDataExd.MesEAppCons);
	                                                                             
	MW_Float( WORD_STRONG := MesBlock_Temp_2[1],  WORD_WEAK := MesBlock_Temp_2[2],  VAR_OUT  := MesDataExd.MesData.MesI1);
	MW_Float( WORD_STRONG := MesBlock_Temp_2[3],  WORD_WEAK := MesBlock_Temp_2[4],  VAR_OUT  := MesDataExd.MesData.MesI2);
	MW_Float( WORD_STRONG := MesBlock_Temp_2[5],  WORD_WEAK := MesBlock_Temp_2[6],  VAR_OUT  := MesDataExd.MesData.MesI3);
	MW_Float( WORD_STRONG := MesBlock_Temp_2[7],  WORD_WEAK := MesBlock_Temp_2[8],  VAR_OUT  := MesDataExd.MesData.MesIn);
	MW_Float( WORD_STRONG := MesBlock_Temp_2[13], WORD_WEAK := MesBlock_Temp_2[14], VAR_OUT  := MesDataExd.MesUnbalanced_I1);
	MW_Float( WORD_STRONG := MesBlock_Temp_2[15], WORD_WEAK := MesBlock_Temp_2[16], VAR_OUT  := MesDataExd.MesUnbalanced_I2);
	MW_Float( WORD_STRONG := MesBlock_Temp_2[17], WORD_WEAK := MesBlock_Temp_2[18], VAR_OUT  := MesDataExd.MesUnbalanced_I3);
	MW_Float( WORD_STRONG := MesBlock_Temp_2[21], WORD_WEAK := MesBlock_Temp_2[22], VAR_OUT  := MesDataExd.MesData.MesU12);
	MW_Float( WORD_STRONG := MesBlock_Temp_2[23], WORD_WEAK := MesBlock_Temp_2[24], VAR_OUT  := MesDataExd.MesData.MesU23);
	MW_Float( WORD_STRONG := MesBlock_Temp_2[25], WORD_WEAK := MesBlock_Temp_2[26], VAR_OUT  := MesDataExd.MesData.MesU31);
	MW_Float( WORD_STRONG := MesBlock_Temp_2[29], WORD_WEAK := MesBlock_Temp_2[30], VAR_OUT  := MesDataExd.MesData.MesV1);
	MW_Float( WORD_STRONG := MesBlock_Temp_2[31], WORD_WEAK := MesBlock_Temp_2[32], VAR_OUT  := MesDataExd.MesData.MesV2);
	MW_Float( WORD_STRONG := MesBlock_Temp_2[33], WORD_WEAK := MesBlock_Temp_2[34], VAR_OUT  := MesDataExd.MesData.MesV3);
	MW_Float( WORD_STRONG := MesBlock_Temp_2[39], WORD_WEAK := MesBlock_Temp_2[40], VAR_OUT  := MesDataExd.MesUnbalanced_U12);
	MW_Float( WORD_STRONG := MesBlock_Temp_2[41], WORD_WEAK := MesBlock_Temp_2[42], VAR_OUT  := MesDataExd.MesUnbalanced_U23);
	MW_Float( WORD_STRONG := MesBlock_Temp_2[43], WORD_WEAK := MesBlock_Temp_2[44], VAR_OUT  := MesDataExd.MesUnbalanced_U31);
	MW_Float( WORD_STRONG := MesBlock_Temp_2[47], WORD_WEAK := MesBlock_Temp_2[48], VAR_OUT  := MesDataExd.MesUnbalanced_V1);
	MW_Float( WORD_STRONG := MesBlock_Temp_2[49], WORD_WEAK := MesBlock_Temp_2[50], VAR_OUT  := MesDataExd.MesUnbalanced_V2);
	MW_Float( WORD_STRONG := MesBlock_Temp_2[51], WORD_WEAK := MesBlock_Temp_2[52], VAR_OUT  := MesDataExd.MesUnbalanced_V3);
	MW_Float( WORD_STRONG := MesBlock_Temp_2[55], WORD_WEAK := MesBlock_Temp_2[56], VAR_OUT  := MesDataExd.MesData.MesP1);
	MW_Float( WORD_STRONG := MesBlock_Temp_2[57], WORD_WEAK := MesBlock_Temp_2[58], VAR_OUT  := MesDataExd.MesData.MesP2);
	MW_Float( WORD_STRONG := MesBlock_Temp_2[59], WORD_WEAK := MesBlock_Temp_2[60], VAR_OUT  := MesDataExd.MesData.MesP3);
	MW_Float( WORD_STRONG := MesBlock_Temp_2[61], WORD_WEAK := MesBlock_Temp_2[62], VAR_OUT  := MesDataExd.MesData.MesP);
	MW_Float( WORD_STRONG := MesBlock_Temp_2[63], WORD_WEAK := MesBlock_Temp_2[64], VAR_OUT  := MesDataExd.MesData.MesQ1);
	MW_Float( WORD_STRONG := MesBlock_Temp_2[65], WORD_WEAK := MesBlock_Temp_2[66], VAR_OUT  := MesDataExd.MesData.MesQ2);
	MW_Float( WORD_STRONG := MesBlock_Temp_2[67], WORD_WEAK := MesBlock_Temp_2[68], VAR_OUT  := MesDataExd.MesData.MesQ3);
	MW_Float( WORD_STRONG := MesBlock_Temp_2[69], WORD_WEAK := MesBlock_Temp_2[70], VAR_OUT  := MesDataExd.MesData.MesQ);
	MW_Float( WORD_STRONG := MesBlock_Temp_2[71], WORD_WEAK := MesBlock_Temp_2[72], VAR_OUT  := MesDataExd.MesData.MesS1);
	MW_Float( WORD_STRONG := MesBlock_Temp_2[73], WORD_WEAK := MesBlock_Temp_2[74], VAR_OUT  := MesDataExd.MesData.MesS2);
	MW_Float( WORD_STRONG := MesBlock_Temp_2[75], WORD_WEAK := MesBlock_Temp_2[76], VAR_OUT  := MesDataExd.MesData.MesS3);
	MW_Float( WORD_STRONG := MesBlock_Temp_2[77], WORD_WEAK := MesBlock_Temp_2[78], VAR_OUT  := MesDataExd.MesData.MesS);
	MW_Float( WORD_STRONG := MesBlock_Temp_2[79], WORD_WEAK := MesBlock_Temp_2[80], VAR_OUT  := MesDataExd.MesData.MesCosPhi1);
	MW_Float( WORD_STRONG := MesBlock_Temp_2[81], WORD_WEAK := MesBlock_Temp_2[82], VAR_OUT  := MesDataExd.MesData.MesCosPhi2);
	MW_Float( WORD_STRONG := MesBlock_Temp_2[83], WORD_WEAK := MesBlock_Temp_2[84], VAR_OUT  := MesDataExd.MesData.MesCosPhi3);
	MW_Float( WORD_STRONG := MesBlock_Temp_2[85], WORD_WEAK := MesBlock_Temp_2[86], VAR_OUT  := MesDataExd.MesData.MesCosPhi);
	MW_Float( WORD_STRONG := MesBlock_Temp_2[111],WORD_WEAK := MesBlock_Temp_2[112],VAR_OUT  := MesDataExd.MesData.MesFreq);

	MW_UInt(WORD_STRONG:= MesBlock_Temp_3[ 1],  VAR_OUT:=MesDataExd.MesAlarmImax);
	MW_UInt(WORD_STRONG:= MesBlock_Temp_3[ 2],  VAR_OUT:=MesDataExd.MesAlarmImin);
	MW_UInt(WORD_STRONG:= MesBlock_Temp_3[ 3],  VAR_OUT:=MesDataExd.MesAlarmInmax);
	MW_UInt(WORD_STRONG:= MesBlock_Temp_3[ 4],  VAR_OUT:=MesDataExd.MesAlarmIgmax);
	MW_UInt(WORD_STRONG:= MesBlock_Temp_3[ 5],  VAR_OUT:=MesDataExd.MesAlarmUmax);
	MW_UInt(WORD_STRONG:= MesBlock_Temp_3[ 6],  VAR_OUT:=MesDataExd.MesAlarmUmin);
	MW_UInt(WORD_STRONG:= MesBlock_Temp_3[ 7],  VAR_OUT:=MesDataExd.MesAlarmVmax);
	MW_UInt(WORD_STRONG:= MesBlock_Temp_3[ 8],  VAR_OUT:=MesDataExd.MesAlarmVmin);
	MW_UInt(WORD_STRONG:= MesBlock_Temp_3[ 9],  VAR_OUT:=MesDataExd.MesAlarmPmax);
	MW_UInt(WORD_STRONG:= MesBlock_Temp_3[ 10], VAR_OUT:=MesDataExd.MesAlarmQmax);
	MW_UInt(WORD_STRONG:= MesBlock_Temp_3[ 11], VAR_OUT:=MesDataExd.MesAlarmSmax);
	
	MW_UInt(WORD_STRONG:= MesBlock_Temp_3[ 25], VAR_OUT:=MesDataExd.MesAlarmFreqmax);
	MW_UInt(WORD_STRONG:= MesBlock_Temp_3[ 26], VAR_OUT:=MesDataExd.MesAlarmFreqmin);
	
	MW_UInt(WORD_STRONG:= MesBlock_Temp_3[ 29], VAR_OUT:=MesDataExd.MesAlarm_PhaseLoss);

	MW_UInt(WORD_STRONG:= MesBlock_Temp_3[ 102], VAR_OUT:=MesDataExd.MesAlarmReset);
	MW_UInt(WORD_STRONG:= MesBlock_Temp_3[ 104], VAR_OUT:=MesDataExd.MesAlarm_PhaseReversal);

END_IF

MesDataExd.MesData.MesI := (MesDataExd.MesData.MesI1 + MesDataExd.MesData.MesI2 + MesDataExd.MesData.MesI3 );
MesDataExd.MesData.MesU := (MesDataExd.MesData.MesU12 + MesDataExd.MesData.MesU23 + MesDataExd.MesData.MesU31 )/3;
MesDataExd.MesData.MesV := (MesDataExd.MesData.MesV1 + MesDataExd.MesData.MesV2 + MesDataExd.MesData.MesV3 )/3;

IF MesDataExd.MesData.MesP <> 0 THEN
	MesDataExd.MesData.MesTanPhi := MesDataExd.MesData.MesQ/MesDataExd.MesData.MesP;
END_IF
END_METHOD

END_FUNCTION_BLOCK

// ---- 01_Equipement_Library/Operation Meter/FB_PM_Prometer.TcPOU
FUNCTION_BLOCK FB_PM_Prometer EXTENDS FB_PM_Base
//////////////////
// Measurement Solution based on Digiware, but access through PMS Socomec
//////////////////
VAR CONSTANT
	// Characteristics of the object (Same for all instances)
			
END_VAR

VAR_INPUT PERSISTENT
	// Parameters of the Object (instance specific) 
	ParamUnitID					: BYTE 		:= 1 ;								// (NA)unit ID
	ParamInInterfaceSub			: BOOL 		:= TRUE; 							// Serial interface RS422/RS485 TYPE (0:EL6021,1:SUB9)
	ParamIPAddress		   		: STRING 	:= '192.168.20.15'; 				// (NA) IP Adress of ION7650 .
	ParamTcpPort				: UINT 		:= 502;					
	
END_VAR

VAR_OUTPUT
	//Child objects
	
END_VAR


VAR_INPUT 
			MesDataExd AT %Q*				: PM_Prometer ;	
END_VAR

VAR
	//M_ALARMMANAGEMENT VARIABLES//
	                                                    								
                                  								

	//M_READ VARIABLES//
		ModbusRead					: ARRAY[1..4] OF FB_ModbusRead ; 		// (NA) FB for Modbus Reading
		ModbusAlarm					: ARRAY[1..4] OF BOOL;					// (NA) Read alarm
		ModbusAlarmsID				: ARRAY[1..4] OF UDINT;					// (NA) Read alarm ID
		MesBlock1_Temp 				: ARRAY[1..4] OF ARRAY[1..125] OF WORD;	// (NA) Temporary Block with multiple modbus reading (U30 + I35)
	
		ObjectCom					: INT;									// (NA) Sequence index
		MesModbusAlarmCode			: UDINT;								// (NA) Modbus Read Alarm Code	
		Busy						: BOOL;
		Error						: BOOL;
		
		
	//M_INIT VARIABLES //
		OutFBCompleteted			: BOOL;
	// M_EXECUTE VARIABLES //

                              

 
END_VAR

METHOD M_AlarmManagement
//////////////////
// Digiware measurement tool alarm and warning management
/////////////////

VAR 
	// Method local variables (reinitialized at each cycle) 
	FB_AlarmCodeManager			: FB_AlarmCodeManager ; 
	
	KK							: BYTE ;		// For loop
	
	CMWarning					: BOOL;			// At least one Digiware device in Alarm
	CMAlarm						: BOOL;			// At least one Digiware device in Alarm
	
END_VAR
CMAlarm := ModbusAlarm[1] AND ModbusAlarm[2];
CMWarning := ModbusAlarm[1] OR ModbusAlarm[2];
	
TON_ComAlarm(IN:= CMAlarm, PT:= ParamTempoComAlarm, Q=>MesComAlarm) ;	
TON_ComWarning(IN:= CMWarning, PT:= ParamTempoComAlarm, Q=>MesComWarning) ;	
//					General com alarm : All the read FB fucked up


// ALARM CODE //
	FB_AlarmCodeManager(
		bAlarm1			:= MesComAlarm  , 					// Communication Error with D50 (= all modules) 
		bAlarm2			:= MesComWarning, 		// 
		bAlarm3			:=FALSE, 		// 
		bAlarm4			:=FALSE, 		// 
		bAlarm5			:=FALSE, 
		bAlarm6			:=FALSE, 
		bAlarm7			:=FALSE, 
		bAlarm8			:=FALSE, 
		bAlarm9			:=FALSE, 
		bAlarm10		:=FALSE, 
		bAlarm11		:=FALSE, 
		bAlarm12		:=FALSE, 
		bAlarm13		:=FALSE, 
		bAlarm14		:=FALSE, 
		bAlarm15		:= FALSE , 			// Command Alarm in case of intervention 							 
		wAlarmCode		=> MesAlarmCode);



// EVENT CODE //
END_METHOD

METHOD M_CP
//////////////////
//  Emulator
/////////////////

VAR 
	// Method local variables (reinitialized at each cycle) 
	
END_VAR


SUPER^.M_CP() ; 




Trig_Cmd_Read(CLK:=IN_CmdToggleRead);
	
IF Trig_Cmd_Read.Q THEN
	IN_CmdToggleRead := FALSE;
	MesDataExd.MesData.MesCP_Read := NOT MesDataExd.MesData.MesCP_Read;
END_IF
END_METHOD

METHOD M_Evaluate : BOOL
VAR_INPUT
END_VAR
MesDataF11.MesAlarmCode 	:= MesAlarmCode;
MesDataF15.MesAlarmCode 	:= MesAlarmCode;
MesDataF21.MesAlarmCode 	:= MesAlarmCode;
MesDataF22.MesAlarmCode 	:= MesAlarmCode;
MesDataT1.MesAlarmCode  	:= MesAlarmCode;
MesDataT2.MesAlarmCode  	:= MesAlarmCode;
MesDataF11.MesWarningCode 	:= MesWarningCode;
MesDataF15.MesWarningCode 	:= MesWarningCode;
MesDataF21.MesWarningCode 	:= MesWarningCode;
MesDataF22.MesWarningCode 	:= MesWarningCode;
MesDataT1.MesWarningCode  	:= MesWarningCode;
MesDataT2.MesWarningCode  	:= MesWarningCode;
END_METHOD

METHOD M_Execute
//////////////////
//  Method Calls 
/////////////////
VAR 
	// Method local variables (reinitialized at each cycle) 
	// EMULATOR
		Psoltot		: REAL;		// Total Solar Power . 
		KK			: BYTE;		// For Loop
	
END_VAR
// READING AND WRITING CLOCK //
	TP1(IN:=NOT TP1.Q , PT:= ParamClockReadTime);
	ClockRead 		:= TP1.Q;

// PERMANENT CONDITIONS //
	CalCP_Read 					:= TRUE  ; 
	
// METHODS CALLS //
	IF bInit THEN
		M_Init() ; 
		bInit					:= FALSE ; 
		
	END_IF

	M_Read() ; 
	M_Evaluate();
// EMULATOR COM READ  /////////////
	
	
	////////////////////
	M_AlarmManagement();
END_METHOD

METHOD M_Read
//////////////////
//  Read Modbus Variable for PCS . 
/////////////////
VAR 
	MW 					: FB_MergeWordsToFloat; 
	KK					: BYTE;  						// FOR Loop 

	AX_Adr				: ARRAY[1..4] OF WORD 		:= [1100,	1200	,250	,260];
	AX_Qty				: ARRAY[1..4] OF WORD		:= [100,	88		,6		,6	];
	AX_UnitID			: ARRAY[1..4] OF BYTE 		:= [1,		1		,1		,1	];

	
	
	mesH: REAL;
END_VAR

// MODBUS REQUEST TCP-IP //
	 
	ModbusRead[1]
	(
		nTcpPort := ParamTcpPort,
		pDestAddr := ADR(MesBlock1_Temp[1]),
		cbLength := SIZEOF(MesBlock1_Temp[1]),
		sIPAddr := ParamIPAddress,
		tTimeout := ParamTimeout,
		nQuantity := AX_Qty[1],
		nMBAddr := AX_Adr[1],
		nUnitID := AX_UnitID[1],
		ClockRead := ClockRead,
		ErrorId => ModbusAlarmsID[1],
		ModbusReadAlarm => ModbusAlarm[1]
	);
	
	ModbusRead[2]
	(
		nTcpPort := ParamTcpPort,
		pDestAddr := ADR(MesBlock1_Temp[2]),
		cbLength := SIZEOF(MesBlock1_Temp[2]),
		sIPAddr := ParamIPAddress,
		tTimeout := ParamTimeout,
		nQuantity := AX_Qty[2],
		nMBAddr := AX_Adr[2],
		nUnitID := AX_UnitID[2],
		ClockRead := ClockRead,
		ErrorId => ModbusAlarmsID[2],
		ModbusReadAlarm => ModbusAlarm[2]
	);
	
	
	ModbusRead[3]
	(
		nTcpPort := ParamTcpPort,
		pDestAddr := ADR(MesBlock1_Temp[3]),
		cbLength := SIZEOF(MesBlock1_Temp[3]),
		sIPAddr := ParamIPAddress,
		tTimeout := ParamTimeout,
		nQuantity := AX_Qty[3],
		nMBAddr := AX_Adr[3],
		nUnitID := AX_UnitID[3],
		ClockRead := ClockRead,
		ErrorId => ModbusAlarmsID[3],
		ModbusReadAlarm => ModbusAlarm[3]
	);				
	ModbusRead[4]
	(
		nTcpPort := ParamTcpPort,
		pDestAddr := ADR(MesBlock1_Temp[4]),
		cbLength := SIZEOF(MesBlock1_Temp[4]),
		sIPAddr := ParamIPAddress,
		tTimeout := ParamTimeout,
		nQuantity := AX_Qty[4],
		nMBAddr := AX_Adr[4],
		nUnitID := AX_UnitID[4],
		ClockRead := ClockRead,
		ErrorId => ModbusAlarmsID[4],
		ModbusReadAlarm => ModbusAlarm[4]
	);	
	// Block 1
	MW(WORD_STRONG := MesBlock1_Temp[1][  2], WORD_WEAK := MesBlock1_Temp[1][  1], VAR_OUT := MesDataExd.T1.MesI1);	
					
